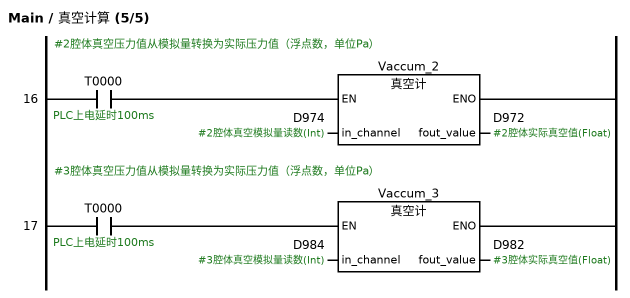
; [picture p24: Main / 真空计算, rungs 16-17]
; rung 16: #2腔体真空压力值从模拟量转换为实际压力值（浮点数，单位Pa）
LD T0000  ; PLC上电延时100ms
CALL Vaccum_2 : 真空计 (in_channel := D974, fout_value => D972)  ; #2腔体真空模拟量读数(Int), #2腔体实际真空值(Float)
; rung 17: #3腔体真空压力值从模拟量转换为实际压力值（浮点数，单位Pa）
LD T0000  ; PLC上电延时100ms
CALL Vaccum_3 : 真空计 (in_channel := D984, fout_value => D982)  ; #3腔体真空模拟量读数(Int), #3腔体实际真空值(Float)

### Section 整机复位

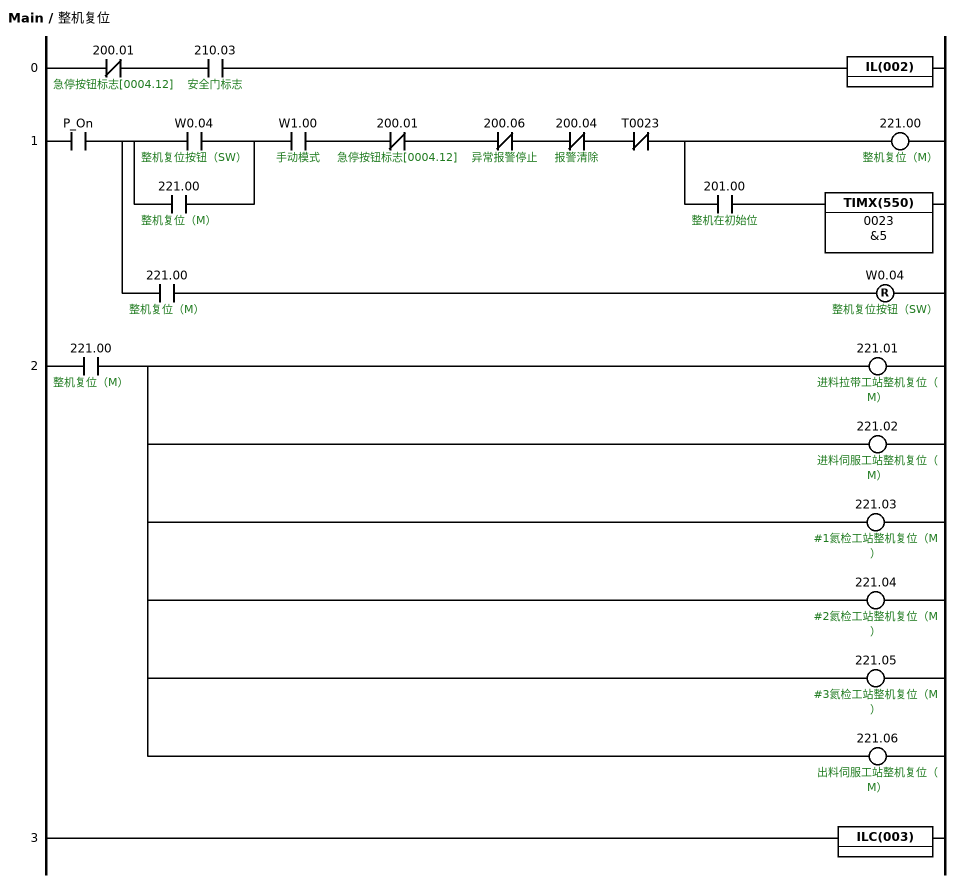
; rung 0
LDNOT 200.01  ; 急停按钮标志[0004.12]
AND 210.03  ; 安全门标志
IL(002)
; rung 1
LD P_On
OUT TR0
LD W0.04  ; 整机复位按钮（SW）
OR 221.00  ; 整机复位（M）
ANDLD
AND W1.00  ; 手动模式
ANDNOT 200.01  ; 急停按钮标志[0004.12]
ANDNOT 200.06  ; 异常报警停止
ANDNOT 200.04  ; 报警清除
ANDNOT T0023
OUT 221.00  ; 整机复位（M）
AND 201.00  ; 整机在初始位
TIMX(550) 0023 &5
LD TR0
AND 221.00  ; 整机复位（M）
RSET W0.04  ; 整机复位按钮（SW）
; rung 2
LD 221.00  ; 整机复位（M）
OUT 221.01  ; 进料拉带工站整机复位（M）
OUT 221.02  ; 进料伺服工站整机复位（M）
OUT 221.03  ; #1氦检工站整机复位（M）
OUT 221.04  ; #2氦检工站整机复位（M）
OUT 221.05  ; #3氦检工站整机复位（M）
OUT 221.06  ; 出料伺服工站整机复位（M）
; rung 3
ILC(003)

### Section 指示灯

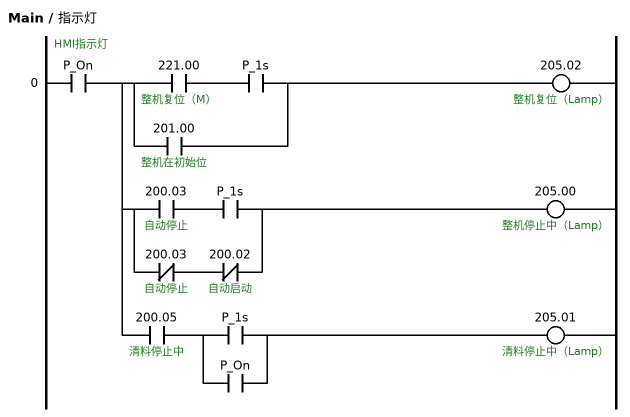
; rung 0: HMI指示灯
LD P_On
OUT TR0
LD 221.00  ; 整机复位（M）
AND P_1s
OR 201.00  ; 整机在初始位
ANDLD
OUT 205.02  ; 整机复位（Lamp）
LD TR0
LD 200.03  ; 自动停止
AND P_1s
LDNOT 200.03  ; 自动停止
ANDNOT 200.02  ; 自动启动
ORLD
ANDLD
OUT 205.00  ; 整机停止中（Lamp）
LD TR0
AND 200.05  ; 清料停止中
LD P_1s
OR P_On
ANDLD
OUT 205.01  ; 清料停止中（Lamp）

### Section 外部输出

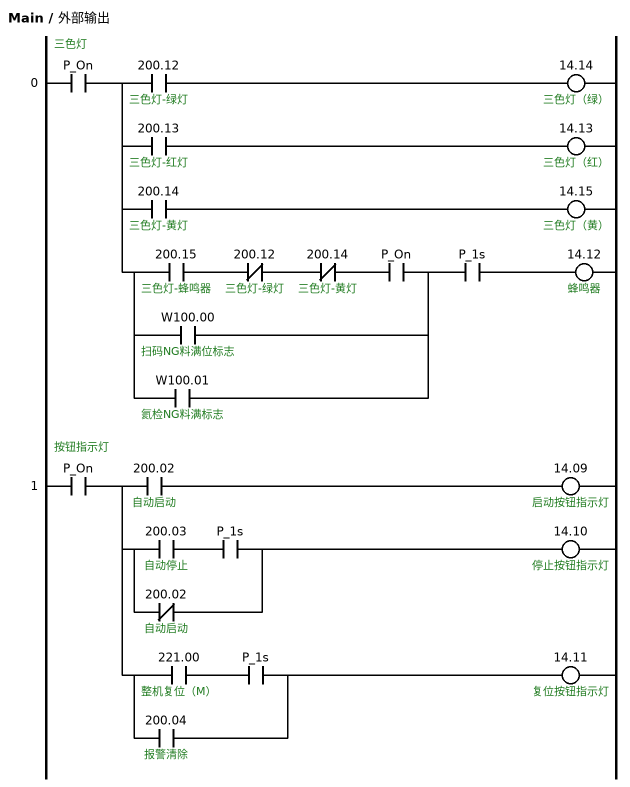
; rung 0: 三色灯
LD P_On
OUT TR0
AND 200.12  ; 三色灯-绿灯
OUT 14.14  ; 三色灯（绿）
LD TR0
AND 200.13  ; 三色灯-红灯
OUT 14.13  ; 三色灯（红）
LD TR0
AND 200.14  ; 三色灯-黄灯
OUT 14.15  ; 三色灯（黄）
LD TR0
LD 200.15  ; 三色灯-蜂鸣器
ANDNOT 200.12  ; 三色灯-绿灯
ANDNOT 200.14  ; 三色灯-黄灯
AND P_On
OR W100.00  ; 扫码NG料满位标志
OR W100.01  ; 氦检NG料满标志
ANDLD
AND P_1s
OUT 14.12  ; 蜂鸣器
; rung 1: 按钮指示灯
LD P_On
OUT TR0
AND 200.02  ; 自动启动
OUT 14.09  ; 启动按钮指示灯
LD TR0
LD 200.03  ; 自动停止
AND P_1s
ORNOT 200.02  ; 自动启动
ANDLD
OUT 14.10  ; 停止按钮指示灯
LD TR0
LD 221.00  ; 整机复位（M）
AND P_1s
OR 200.04  ; 报警清除
ANDLD
OUT 14.11  ; 复位按钮指示灯

### Section END
; rung 0
END(001)

## Program 进料拉带机构 (cyclic task 1)

### Section Main

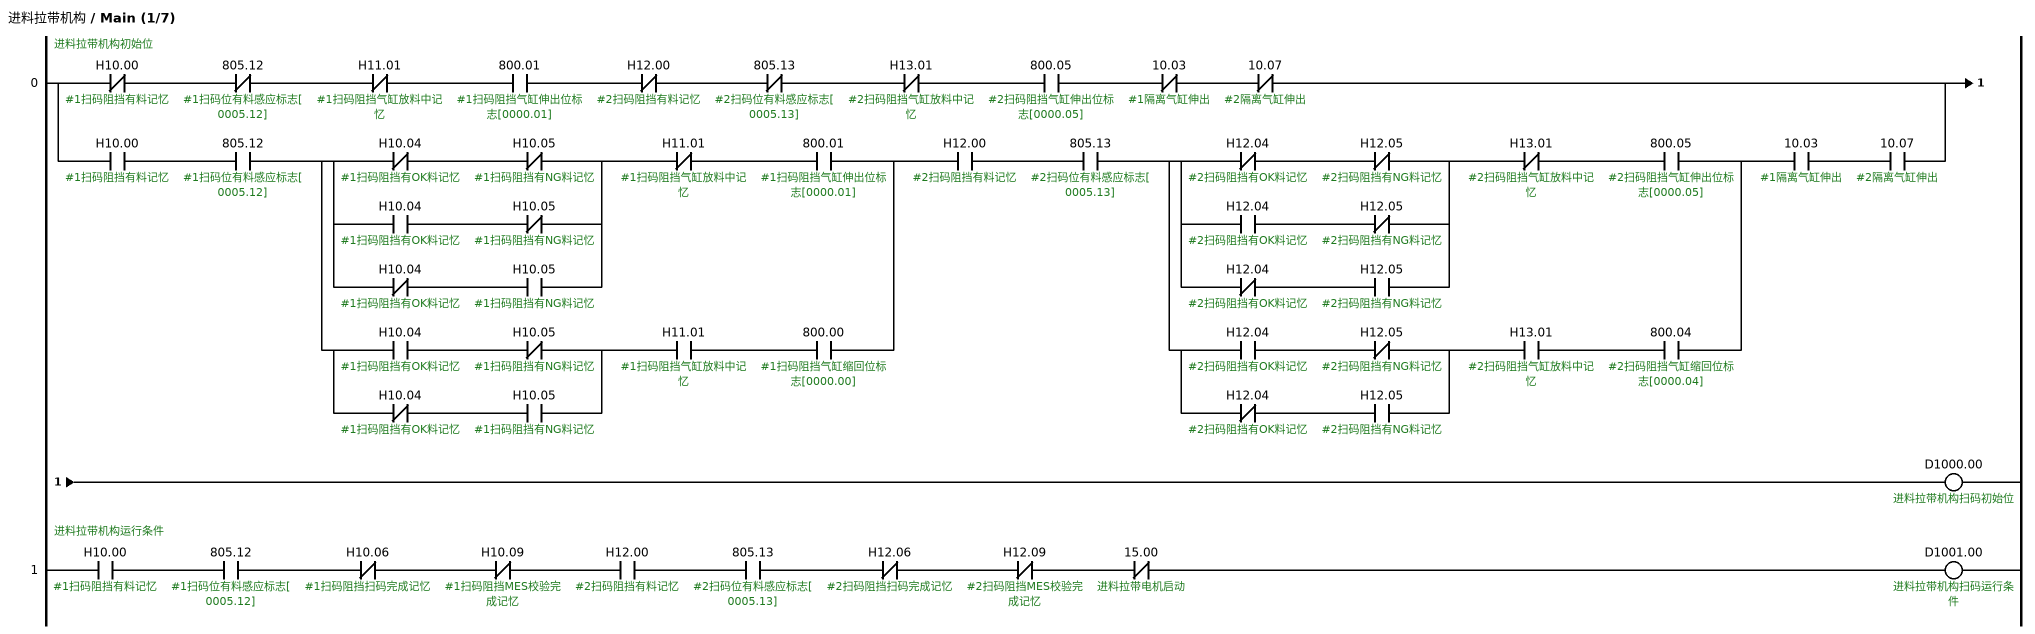
; rung 0: 进料拉带机构初始位
LDNOT H10.00  ; #1扫码阻挡有料记忆
ANDNOT 805.12  ; #1扫码位有料感应标志[0005.12]
ANDNOT H11.01  ; #1扫码阻挡气缸放料中记忆
AND 800.01  ; #1扫码阻挡气缸伸出位标志[0000.01]
ANDNOT H12.00  ; #2扫码阻挡有料记忆
ANDNOT 805.13  ; #2扫码位有料感应标志[0005.13]
ANDNOT H13.01  ; #2扫码阻挡气缸放料中记忆
AND 800.05  ; #2扫码阻挡气缸伸出位标志[0000.05]
ANDNOT 10.03  ; #1隔离气缸伸出
ANDNOT 10.07  ; #2隔离气缸伸出
LD H10.00  ; #1扫码阻挡有料记忆
AND 805.12  ; #1扫码位有料感应标志[0005.12]
LDNOT H10.04  ; #1扫码阻挡有OK料记忆
ANDNOT H10.05  ; #1扫码阻挡有NG料记忆
LD H10.04  ; #1扫码阻挡有OK料记忆
ANDNOT H10.05  ; #1扫码阻挡有NG料记忆
ORLD
LDNOT H10.04  ; #1扫码阻挡有OK料记忆
AND H10.05  ; #1扫码阻挡有NG料记忆
ORLD
ANDNOT H11.01  ; #1扫码阻挡气缸放料中记忆
AND 800.01  ; #1扫码阻挡气缸伸出位标志[0000.01]
LD H10.04  ; #1扫码阻挡有OK料记忆
ANDNOT H10.05  ; #1扫码阻挡有NG料记忆
LDNOT H10.04  ; #1扫码阻挡有OK料记忆
AND H10.05  ; #1扫码阻挡有NG料记忆
ORLD
AND H11.01  ; #1扫码阻挡气缸放料中记忆
AND 800.00  ; #1扫码阻挡气缸缩回位标志[0000.00]
ORLD
ANDLD
AND H12.00  ; #2扫码阻挡有料记忆
AND 805.13  ; #2扫码位有料感应标志[0005.13]
LDNOT H12.04  ; #2扫码阻挡有OK料记忆
ANDNOT H12.05  ; #2扫码阻挡有NG料记忆
LD H12.04  ; #2扫码阻挡有OK料记忆
ANDNOT H12.05  ; #2扫码阻挡有NG料记忆
ORLD
LDNOT H12.04  ; #2扫码阻挡有OK料记忆
AND H12.05  ; #2扫码阻挡有NG料记忆
ORLD
ANDNOT H13.01  ; #2扫码阻挡气缸放料中记忆
AND 800.05  ; #2扫码阻挡气缸伸出位标志[0000.05]
LD H12.04  ; #2扫码阻挡有OK料记忆
ANDNOT H12.05  ; #2扫码阻挡有NG料记忆
LDNOT H12.04  ; #2扫码阻挡有OK料记忆
AND H12.05  ; #2扫码阻挡有NG料记忆
ORLD
AND H13.01  ; #2扫码阻挡气缸放料中记忆
AND 800.04  ; #2扫码阻挡气缸缩回位标志[0000.04]
ORLD
ANDLD
AND 10.03  ; #1隔离气缸伸出
AND 10.07  ; #2隔离气缸伸出
ORLD
OUT D1000.00  ; 进料拉带机构扫码初始位
; rung 1: 进料拉带机构运行条件
LD H10.00  ; #1扫码阻挡有料记忆
AND 805.12  ; #1扫码位有料感应标志[0005.12]
ANDNOT H10.06  ; #1扫码阻挡扫码完成记忆
ANDNOT H10.09  ; #1扫码阻挡MES校验完成记忆
AND H12.00  ; #2扫码阻挡有料记忆
AND 805.13  ; #2扫码位有料感应标志[0005.13]
ANDNOT H12.06  ; #2扫码阻挡扫码完成记忆
ANDNOT H12.09  ; #2扫码阻挡MES校验完成记忆
ANDNOT 15.00  ; 进料拉带电机启动
OUT D1001.00  ; 进料拉带机构扫码运行条件

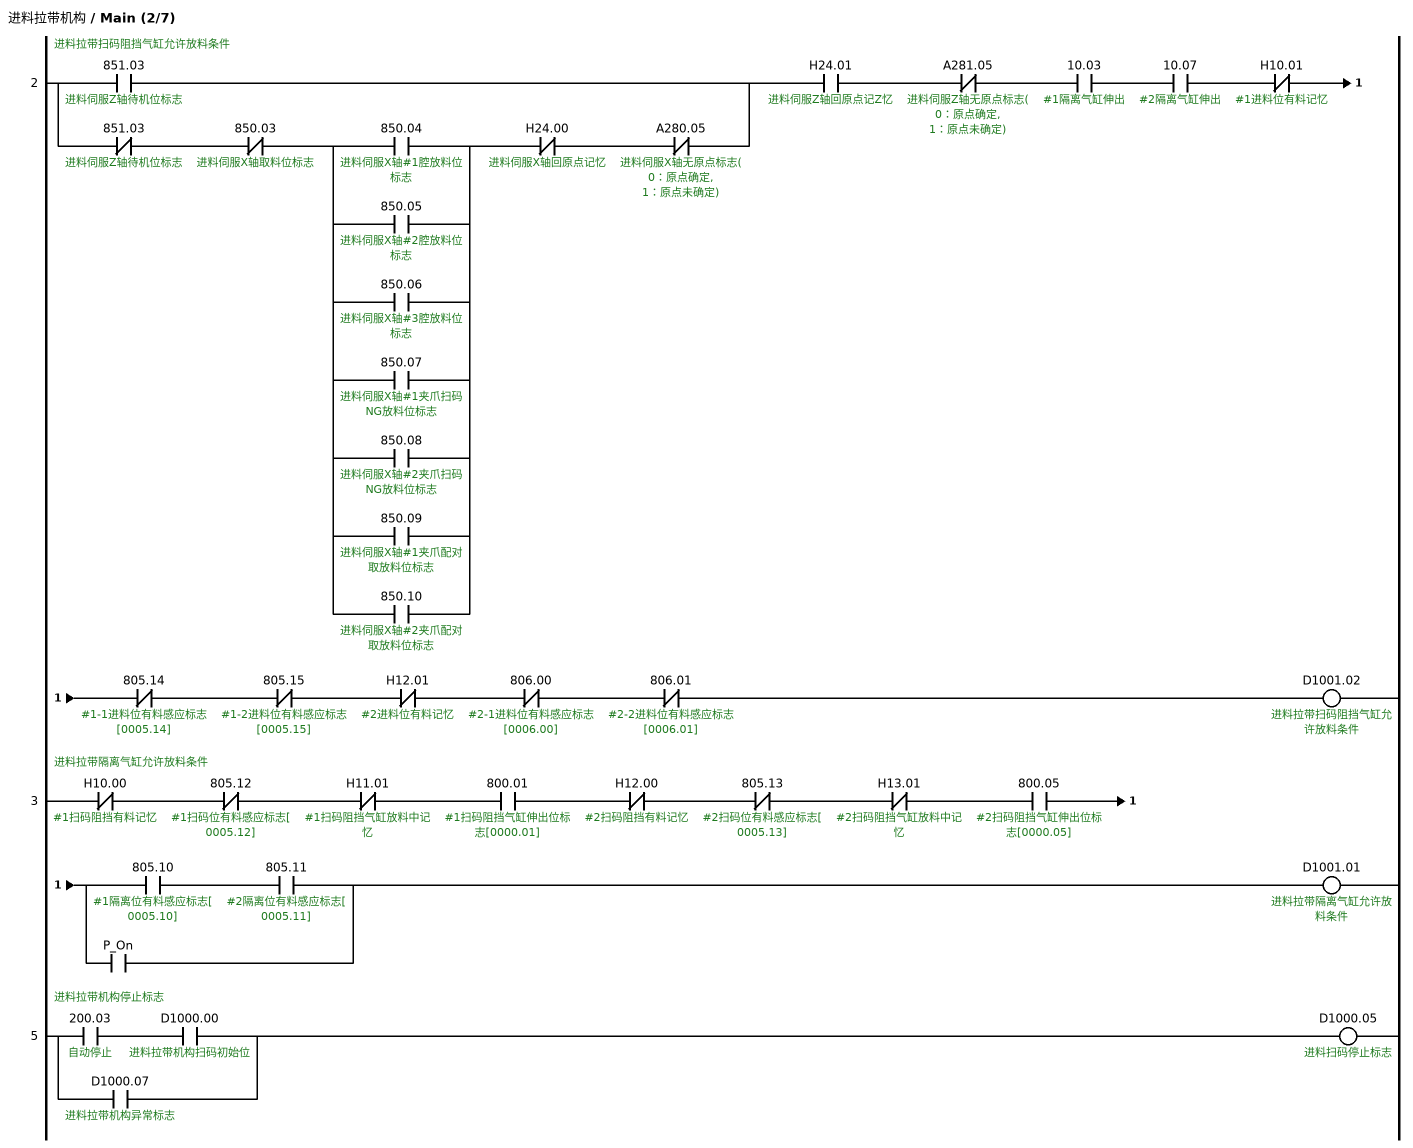
; rung 2: 进料拉带扫码阻挡气缸允许放料条件
LD 851.03  ; 进料伺服Z轴待机位标志
LDNOT 851.03  ; 进料伺服Z轴待机位标志
ANDNOT 850.03  ; 进料伺服X轴取料位标志
LD 850.04  ; 进料伺服X轴#1腔放料位标志
OR 850.05  ; 进料伺服X轴#2腔放料位标志
OR 850.06  ; 进料伺服X轴#3腔放料位标志
OR 850.07  ; 进料伺服X轴#1夹爪扫码NG放料位标志
OR 850.08  ; 进料伺服X轴#2夹爪扫码NG放料位标志
OR 850.09  ; 进料伺服X轴#1夹爪配对取放料位标志
OR 850.10  ; 进料伺服X轴#2夹爪配对取放料位标志
ANDLD
ANDNOT H24.00  ; 进料伺服X轴回原点记忆
ANDNOT A280.05  ; 进料伺服X轴无原点标志(0：原点确定,1：原点未确定)
ORLD
AND H24.01  ; 进料伺服Z轴回原点记Z忆
ANDNOT A281.05  ; 进料伺服Z轴无原点标志(0：原点确定,1：原点未确定)
AND 10.03  ; #1隔离气缸伸出
AND 10.07  ; #2隔离气缸伸出
ANDNOT H10.01  ; #1进料位有料记忆
ANDNOT 805.14  ; #1-1进料位有料感应标志[0005.14]
ANDNOT 805.15  ; #1-2进料位有料感应标志[0005.15]
ANDNOT H12.01  ; #2进料位有料记忆
ANDNOT 806.00  ; #2-1进料位有料感应标志[0006.00]
ANDNOT 806.01  ; #2-2进料位有料感应标志[0006.01]
OUT D1001.02  ; 进料拉带扫码阻挡气缸允许放料条件
; rung 3: 进料拉带隔离气缸允许放料条件
LDNOT H10.00  ; #1扫码阻挡有料记忆
ANDNOT 805.12  ; #1扫码位有料感应标志[0005.12]
ANDNOT H11.01  ; #1扫码阻挡气缸放料中记忆
AND 800.01  ; #1扫码阻挡气缸伸出位标志[0000.01]
ANDNOT H12.00  ; #2扫码阻挡有料记忆
ANDNOT 805.13  ; #2扫码位有料感应标志[0005.13]
ANDNOT H13.01  ; #2扫码阻挡气缸放料中记忆
AND 800.05  ; #2扫码阻挡气缸伸出位标志[0000.05]
LD 805.10  ; #1隔离位有料感应标志[0005.10]
AND 805.11  ; #2隔离位有料感应标志[0005.11]
OR P_On
ANDLD
OUT D1001.01  ; 进料拉带隔离气缸允许放料条件
; rung 4: 进料拉带上料位允许抓料条件
; rung 5: 进料拉带机构停止标志
LD 200.03  ; 自动停止
AND D1000.00  ; 进料拉带机构扫码初始位
OR D1000.07  ; 进料拉带机构异常标志
OUT D1000.05  ; 进料扫码停止标志

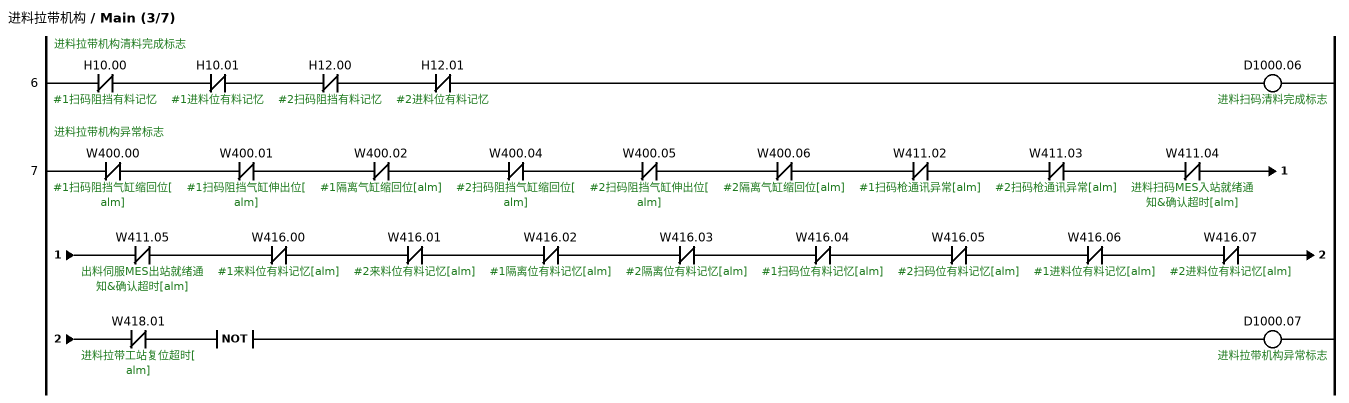
; rung 6: 进料拉带机构清料完成标志
LDNOT H10.00  ; #1扫码阻挡有料记忆
ANDNOT H10.01  ; #1进料位有料记忆
ANDNOT H12.00  ; #2扫码阻挡有料记忆
ANDNOT H12.01  ; #2进料位有料记忆
OUT D1000.06  ; 进料扫码清料完成标志
; rung 7: 进料拉带机构异常标志
LDNOT W400.00  ; #1扫码阻挡气缸缩回位[alm]
ANDNOT W400.01  ; #1扫码阻挡气缸伸出位[alm]
ANDNOT W400.02  ; #1隔离气缸缩回位[alm]
ANDNOT W400.04  ; #2扫码阻挡气缸缩回位[alm]
ANDNOT W400.05  ; #2扫码阻挡气缸伸出位[alm]
ANDNOT W400.06  ; #2隔离气缸缩回位[alm]
ANDNOT W411.02  ; #1扫码枪通讯异常[alm]
ANDNOT W411.03  ; #2扫码枪通讯异常[alm]
ANDNOT W411.04  ; 进料扫码MES入站就绪通知&确认超时[alm]
ANDNOT W411.05  ; 出料伺服MES出站就绪通知&确认超时[alm]
ANDNOT W416.00  ; #1来料位有料记忆[alm]
ANDNOT W416.01  ; #2来料位有料记忆[alm]
ANDNOT W416.02  ; #1隔离位有料记忆[alm]
ANDNOT W416.03  ; #2隔离位有料记忆[alm]
ANDNOT W416.04  ; #1扫码位有料记忆[alm]
ANDNOT W416.05  ; #2扫码位有料记忆[alm]
ANDNOT W416.06  ; #1进料位有料记忆[alm]
ANDNOT W416.07  ; #2进料位有料记忆[alm]
ANDNOT W418.01  ; 进料拉带工站复位超时[alm]
NOT(520)
OUT D1000.07  ; 进料拉带机构异常标志

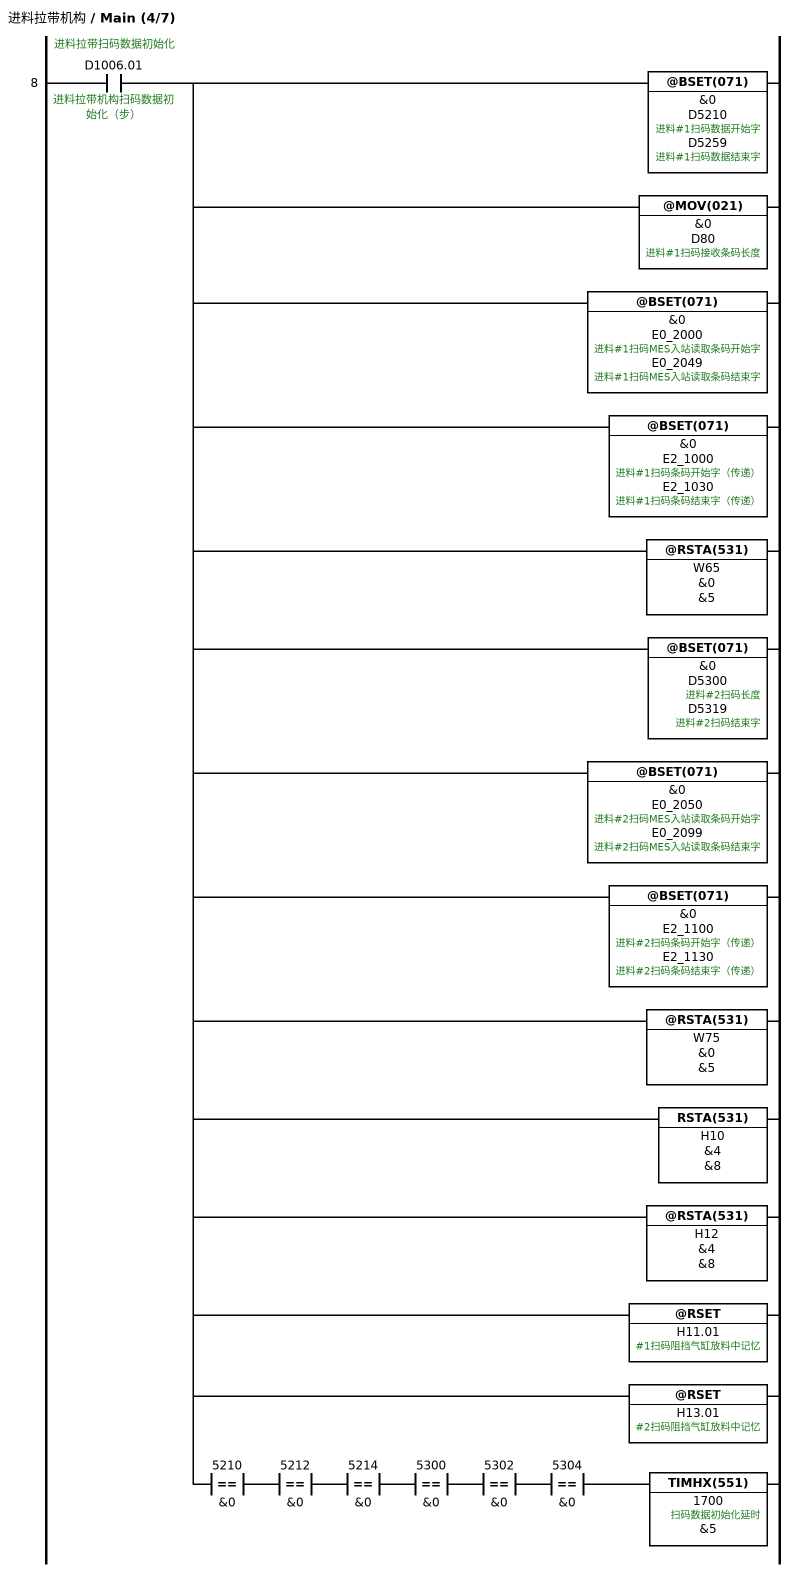
; rung 8: 进料拉带扫码数据初始化
LD D1006.01  ; 进料拉带机构扫码数据初始化（步）
@BSET(071) &0 D5210 D5259  ; 进料#1扫码数据开始字, 进料#1扫码数据结束字
@MOV(021) &0 D80  ; 进料#1扫码接收条码长度
@BSET(071) &0 E0_2000 E0_2049  ; 进料#1扫码MES入站读取条码开始字, 进料#1扫码MES入站读取条码结束字
@BSET(071) &0 E2_1000 E2_1030  ; 进料#1扫码条码开始字（传递）, 进料#1扫码条码结束字（传递）
@RSTA(531) W65 &0 &5
@BSET(071) &0 D5300 D5319  ; 进料#2扫码长度, 进料#2扫码结束字
@BSET(071) &0 E0_2050 E0_2099  ; 进料#2扫码MES入站读取条码开始字, 进料#2扫码MES入站读取条码结束字
@BSET(071) &0 E2_1100 E2_1130  ; 进料#2扫码条码开始字（传递）, 进料#2扫码条码结束字（传递）
@RSTA(531) W75 &0 &5
RSTA(531) H10 &4 &8
@RSTA(531) H12 &4 &8
@RSET H11.01  ; #1扫码阻挡气缸放料中记忆
@RSET H13.01  ; #2扫码阻挡气缸放料中记忆
AND=L(301) 5210 &0
AND=L(301) 5212 &0
AND=L(301) 5214 &0
AND=L(301) 5300 &0
AND=L(301) 5302 &0
AND=L(301) 5304 &0
TIMHX(551) 1700 &5  ; 扫码数据初始化延时

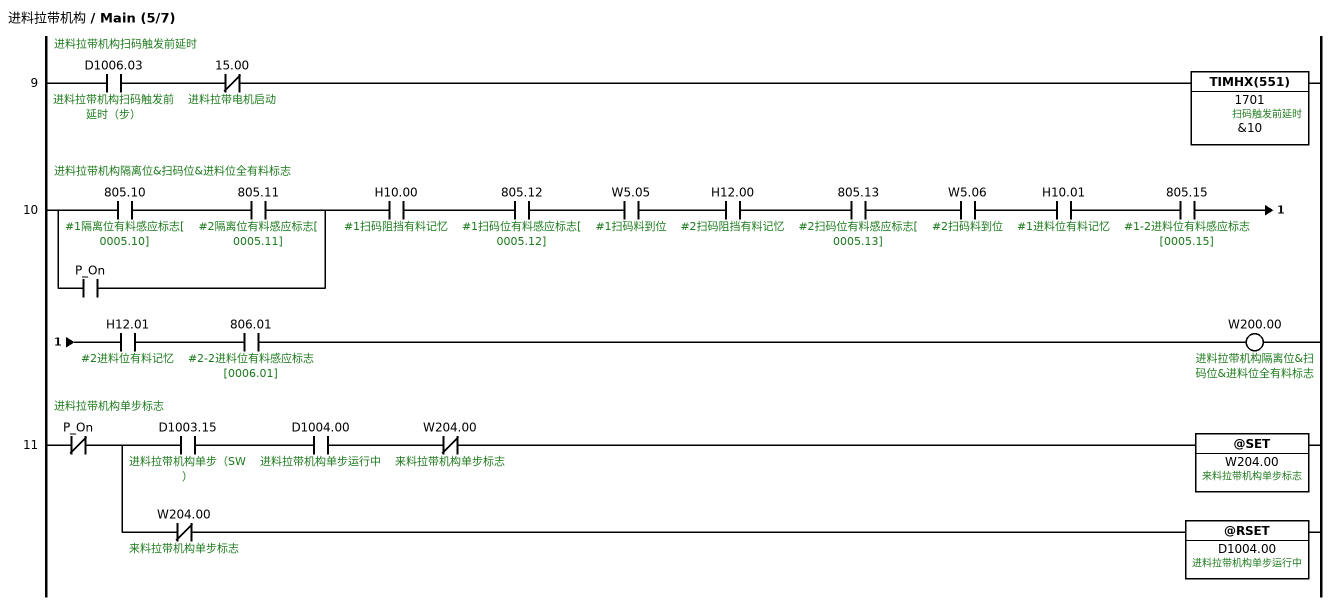
; rung 9: 进料拉带机构扫码触发前延时
LD D1006.03  ; 进料拉带机构扫码触发前延时（步）
ANDNOT 15.00  ; 进料拉带电机启动
TIMHX(551) 1701 &10  ; 扫码触发前延时
; rung 10: 进料拉带机构隔离位&扫码位&进料位全有料标志
LD 805.10  ; #1隔离位有料感应标志[0005.10]
AND 805.11  ; #2隔离位有料感应标志[0005.11]
OR P_On
AND H10.00  ; #1扫码阻挡有料记忆
AND 805.12  ; #1扫码位有料感应标志[0005.12]
AND W5.05  ; #1扫码料到位
AND H12.00  ; #2扫码阻挡有料记忆
AND 805.13  ; #2扫码位有料感应标志[0005.13]
AND W5.06  ; #2扫码料到位
AND H10.01  ; #1进料位有料记忆
AND 805.15  ; #1-2进料位有料感应标志[0005.15]
AND H12.01  ; #2进料位有料记忆
AND 806.01  ; #2-2进料位有料感应标志[0006.01]
OUT W200.00  ; 进料拉带机构隔离位&扫码位&进料位全有料标志
; rung 11: 进料拉带机构单步标志
LDNOT P_On
OUT TR0
AND D1003.15  ; 进料拉带机构单步（SW）
AND D1004.00  ; 进料拉带机构单步运行中
ANDNOT W204.00  ; 来料拉带机构单步标志
@SET W204.00  ; 来料拉带机构单步标志
LD TR0
ANDNOT W204.00  ; 来料拉带机构单步标志
@RSET D1004.00  ; 进料拉带机构单步运行中

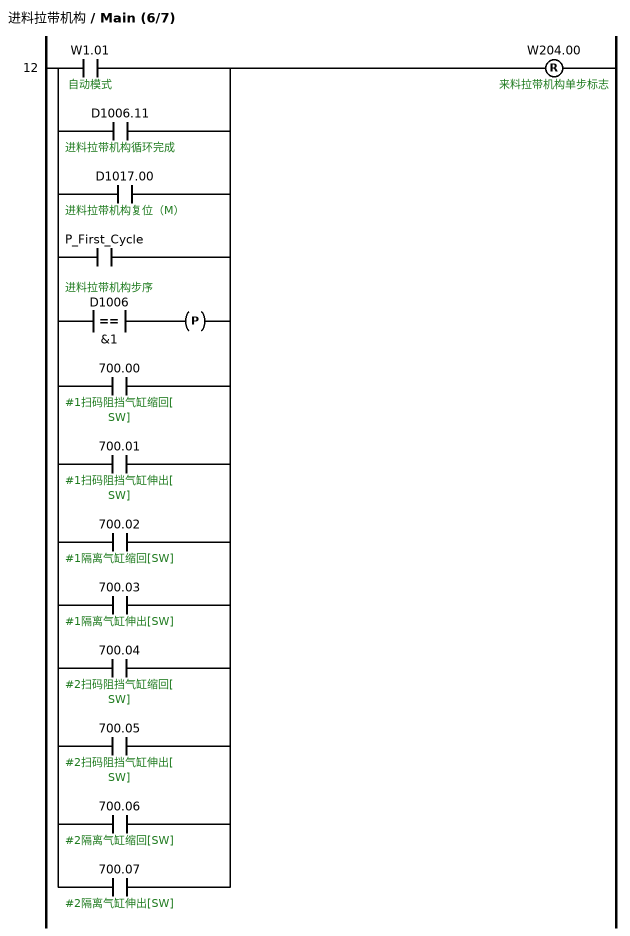
; rung 12
LD W1.01  ; 自动模式
OR D1006.11  ; 进料拉带机构循环完成
OR D1017.00  ; 进料拉带机构复位（M）
OR P_First_Cycle
LD=(300) D1006 &1  ; 进料拉带机构步序
UP(521)
ORLD
OR 700.00  ; #1扫码阻挡气缸缩回[SW]
OR 700.01  ; #1扫码阻挡气缸伸出[SW]
OR 700.02  ; #1隔离气缸缩回[SW]
OR 700.03  ; #1隔离气缸伸出[SW]
OR 700.04  ; #2扫码阻挡气缸缩回[SW]
OR 700.05  ; #2扫码阻挡气缸伸出[SW]
OR 700.06  ; #2隔离气缸缩回[SW]
OR 700.07  ; #2隔离气缸伸出[SW]
RSET W204.00  ; 来料拉带机构单步标志

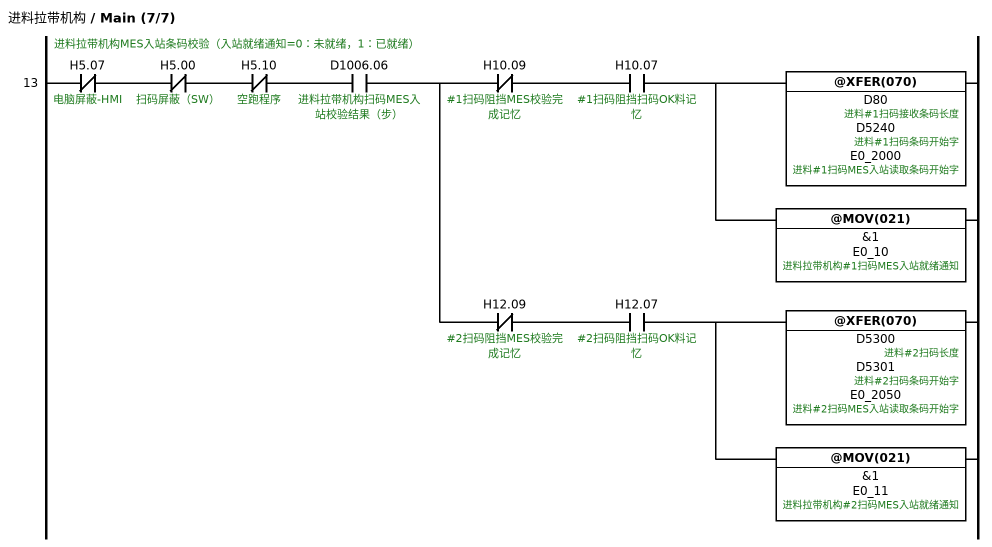
; rung 13: 进料拉带机构MES入站条码校验（入站就绪通知=0：未就绪，1：已就绪）
LDNOT H5.07  ; 电脑屏蔽-HMI
ANDNOT H5.00  ; 扫码屏蔽（SW）
ANDNOT H5.10  ; 空跑程序
AND D1006.06  ; 进料拉带机构扫码MES入站校验结果（步）
OUT TR0
ANDNOT H10.09  ; #1扫码阻挡MES校验完成记忆
AND H10.07  ; #1扫码阻挡扫码OK料记忆
@XFER(070) D80 D5240 E0_2000  ; 进料#1扫码接收条码长度, 进料#1扫码条码开始字, 进料#1扫码MES入站读取条码开始字
@MOV(021) &1 E0_10  ; 进料拉带机构#1扫码MES入站就绪通知
LD TR0
ANDNOT H12.09  ; #2扫码阻挡MES校验完成记忆
AND H12.07  ; #2扫码阻挡扫码OK料记忆
@XFER(070) D5300 D5301 E0_2050  ; 进料#2扫码长度, 进料#2扫码条码开始字, 进料#2扫码MES入站读取条码开始字
@MOV(021) &1 E0_11  ; 进料拉带机构#2扫码MES入站就绪通知

### Section 进料手动

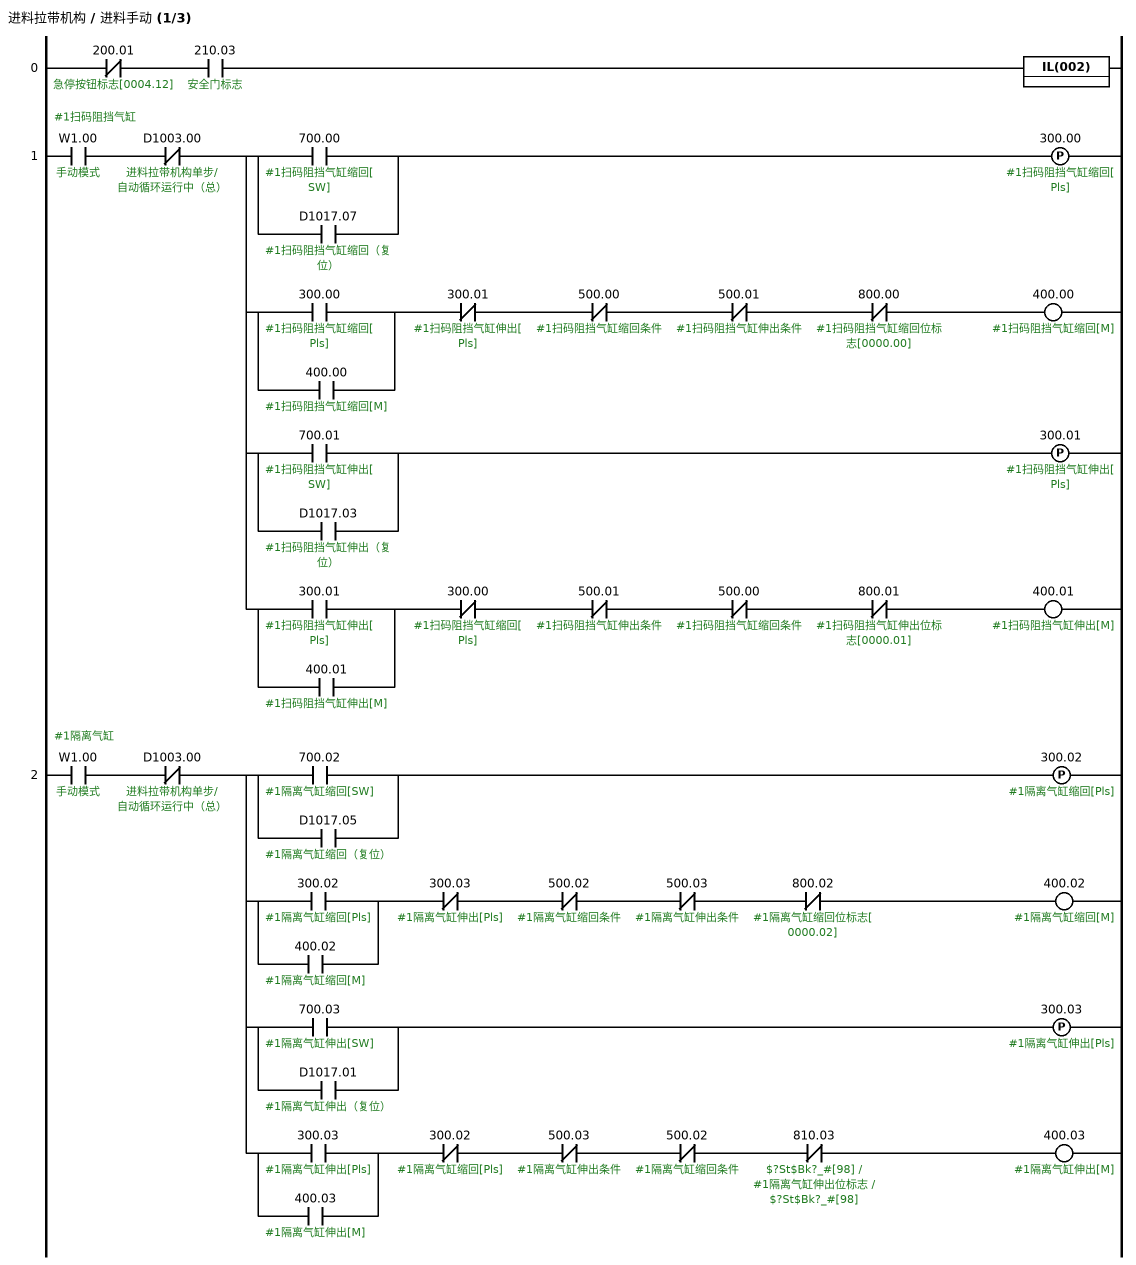
; rung 0
LDNOT 200.01  ; 急停按钮标志[0004.12]
AND 210.03  ; 安全门标志
IL(002)
; rung 1: #1扫码阻挡气缸
LD W1.00  ; 手动模式
ANDNOT D1003.00  ; 进料拉带机构单步/自动循环运行中（总）
OUT TR0
LD 700.00  ; #1扫码阻挡气缸缩回[SW]
OR D1017.07  ; #1扫码阻挡气缸缩回（复位）
ANDLD
DIFU(013) 300.00  ; #1扫码阻挡气缸缩回[Pls]
LD TR0
LD 300.00  ; #1扫码阻挡气缸缩回[Pls]
OR 400.00  ; #1扫码阻挡气缸缩回[M]
ANDLD
ANDNOT 300.01  ; #1扫码阻挡气缸伸出[Pls]
ANDNOT 500.00  ; #1扫码阻挡气缸缩回条件
ANDNOT 500.01  ; #1扫码阻挡气缸伸出条件
ANDNOT 800.00  ; #1扫码阻挡气缸缩回位标志[0000.00]
OUT 400.00  ; #1扫码阻挡气缸缩回[M]
LD TR0
LD 700.01  ; #1扫码阻挡气缸伸出[SW]
OR D1017.03  ; #1扫码阻挡气缸伸出（复位）
ANDLD
DIFU(013) 300.01  ; #1扫码阻挡气缸伸出[Pls]
LD TR0
LD 300.01  ; #1扫码阻挡气缸伸出[Pls]
OR 400.01  ; #1扫码阻挡气缸伸出[M]
ANDLD
ANDNOT 300.00  ; #1扫码阻挡气缸缩回[Pls]
ANDNOT 500.01  ; #1扫码阻挡气缸伸出条件
ANDNOT 500.00  ; #1扫码阻挡气缸缩回条件
ANDNOT 800.01  ; #1扫码阻挡气缸伸出位标志[0000.01]
OUT 400.01  ; #1扫码阻挡气缸伸出[M]
; rung 2: #1隔离气缸
LD W1.00  ; 手动模式
ANDNOT D1003.00  ; 进料拉带机构单步/自动循环运行中（总）
OUT TR0
LD 700.02  ; #1隔离气缸缩回[SW]
OR D1017.05  ; #1隔离气缸缩回（复位）
ANDLD
DIFU(013) 300.02  ; #1隔离气缸缩回[Pls]
LD TR0
LD 300.02  ; #1隔离气缸缩回[Pls]
OR 400.02  ; #1隔离气缸缩回[M]
ANDLD
ANDNOT 300.03  ; #1隔离气缸伸出[Pls]
ANDNOT 500.02  ; #1隔离气缸缩回条件
ANDNOT 500.03  ; #1隔离气缸伸出条件
ANDNOT 800.02  ; #1隔离气缸缩回位标志[0000.02]
OUT 400.02  ; #1隔离气缸缩回[M]
LD TR0
LD 700.03  ; #1隔离气缸伸出[SW]
OR D1017.01  ; #1隔离气缸伸出（复位）
ANDLD
DIFU(013) 300.03  ; #1隔离气缸伸出[Pls]
LD TR0
LD 300.03  ; #1隔离气缸伸出[Pls]
OR 400.03  ; #1隔离气缸伸出[M]
ANDLD
ANDNOT 300.02  ; #1隔离气缸缩回[Pls]
ANDNOT 500.03  ; #1隔离气缸伸出条件
ANDNOT 500.02  ; #1隔离气缸缩回条件
ANDNOT 810.03  ; $?St$Bk?_#[98] / #1隔离气缸伸出位标志 / $?St$Bk?_#[98]
OUT 400.03  ; #1隔离气缸伸出[M]

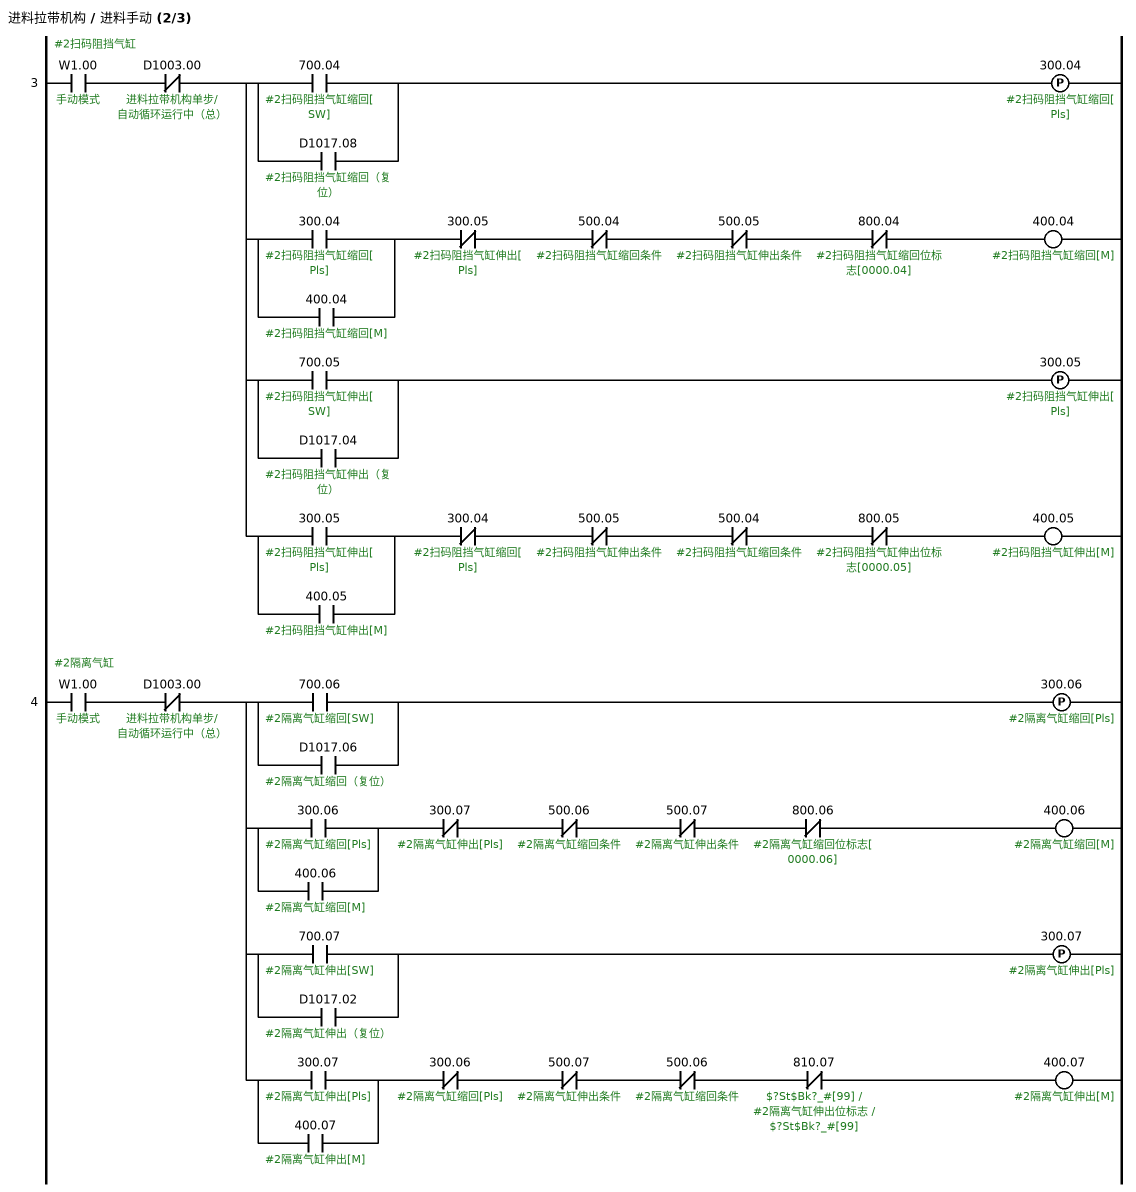
; rung 3: #2扫码阻挡气缸
LD W1.00  ; 手动模式
ANDNOT D1003.00  ; 进料拉带机构单步/自动循环运行中（总）
OUT TR0
LD 700.04  ; #2扫码阻挡气缸缩回[SW]
OR D1017.08  ; #2扫码阻挡气缸缩回（复位）
ANDLD
DIFU(013) 300.04  ; #2扫码阻挡气缸缩回[Pls]
LD TR0
LD 300.04  ; #2扫码阻挡气缸缩回[Pls]
OR 400.04  ; #2扫码阻挡气缸缩回[M]
ANDLD
ANDNOT 300.05  ; #2扫码阻挡气缸伸出[Pls]
ANDNOT 500.04  ; #2扫码阻挡气缸缩回条件
ANDNOT 500.05  ; #2扫码阻挡气缸伸出条件
ANDNOT 800.04  ; #2扫码阻挡气缸缩回位标志[0000.04]
OUT 400.04  ; #2扫码阻挡气缸缩回[M]
LD TR0
LD 700.05  ; #2扫码阻挡气缸伸出[SW]
OR D1017.04  ; #2扫码阻挡气缸伸出（复位）
ANDLD
DIFU(013) 300.05  ; #2扫码阻挡气缸伸出[Pls]
LD TR0
LD 300.05  ; #2扫码阻挡气缸伸出[Pls]
OR 400.05  ; #2扫码阻挡气缸伸出[M]
ANDLD
ANDNOT 300.04  ; #2扫码阻挡气缸缩回[Pls]
ANDNOT 500.05  ; #2扫码阻挡气缸伸出条件
ANDNOT 500.04  ; #2扫码阻挡气缸缩回条件
ANDNOT 800.05  ; #2扫码阻挡气缸伸出位标志[0000.05]
OUT 400.05  ; #2扫码阻挡气缸伸出[M]
; rung 4: #2隔离气缸
LD W1.00  ; 手动模式
ANDNOT D1003.00  ; 进料拉带机构单步/自动循环运行中（总）
OUT TR0
LD 700.06  ; #2隔离气缸缩回[SW]
OR D1017.06  ; #2隔离气缸缩回（复位）
ANDLD
DIFU(013) 300.06  ; #2隔离气缸缩回[Pls]
LD TR0
LD 300.06  ; #2隔离气缸缩回[Pls]
OR 400.06  ; #2隔离气缸缩回[M]
ANDLD
ANDNOT 300.07  ; #2隔离气缸伸出[Pls]
ANDNOT 500.06  ; #2隔离气缸缩回条件
ANDNOT 500.07  ; #2隔离气缸伸出条件
ANDNOT 800.06  ; #2隔离气缸缩回位标志[0000.06]
OUT 400.06  ; #2隔离气缸缩回[M]
LD TR0
LD 700.07  ; #2隔离气缸伸出[SW]
OR D1017.02  ; #2隔离气缸伸出（复位）
ANDLD
DIFU(013) 300.07  ; #2隔离气缸伸出[Pls]
LD TR0
LD 300.07  ; #2隔离气缸伸出[Pls]
OR 400.07  ; #2隔离气缸伸出[M]
ANDLD
ANDNOT 300.06  ; #2隔离气缸缩回[Pls]
ANDNOT 500.07  ; #2隔离气缸伸出条件
ANDNOT 500.06  ; #2隔离气缸缩回条件
ANDNOT 810.07  ; $?St$Bk?_#[99] / #2隔离气缸伸出位标志 / $?St$Bk?_#[99]
OUT 400.07  ; #2隔离气缸伸出[M]

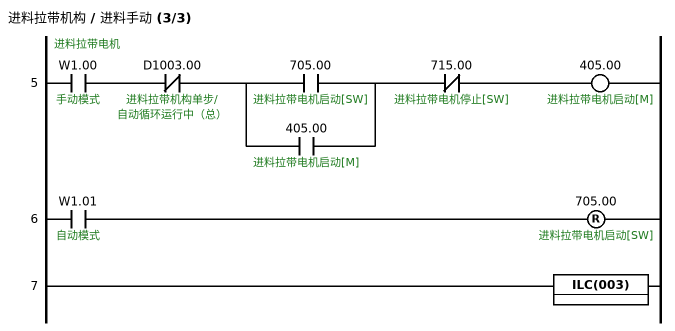
; rung 5: 进料拉带电机
LD W1.00  ; 手动模式
ANDNOT D1003.00  ; 进料拉带机构单步/自动循环运行中（总）
LD 705.00  ; 进料拉带电机启动[SW]
OR 405.00  ; 进料拉带电机启动[M]
ANDLD
ANDNOT 715.00  ; 进料拉带电机停止[SW]
OUT 405.00  ; 进料拉带电机启动[M]
; rung 6
LD W1.01  ; 自动模式
RSET 705.00  ; 进料拉带电机启动[SW]
; rung 7
ILC(003)

### Section 进料自动

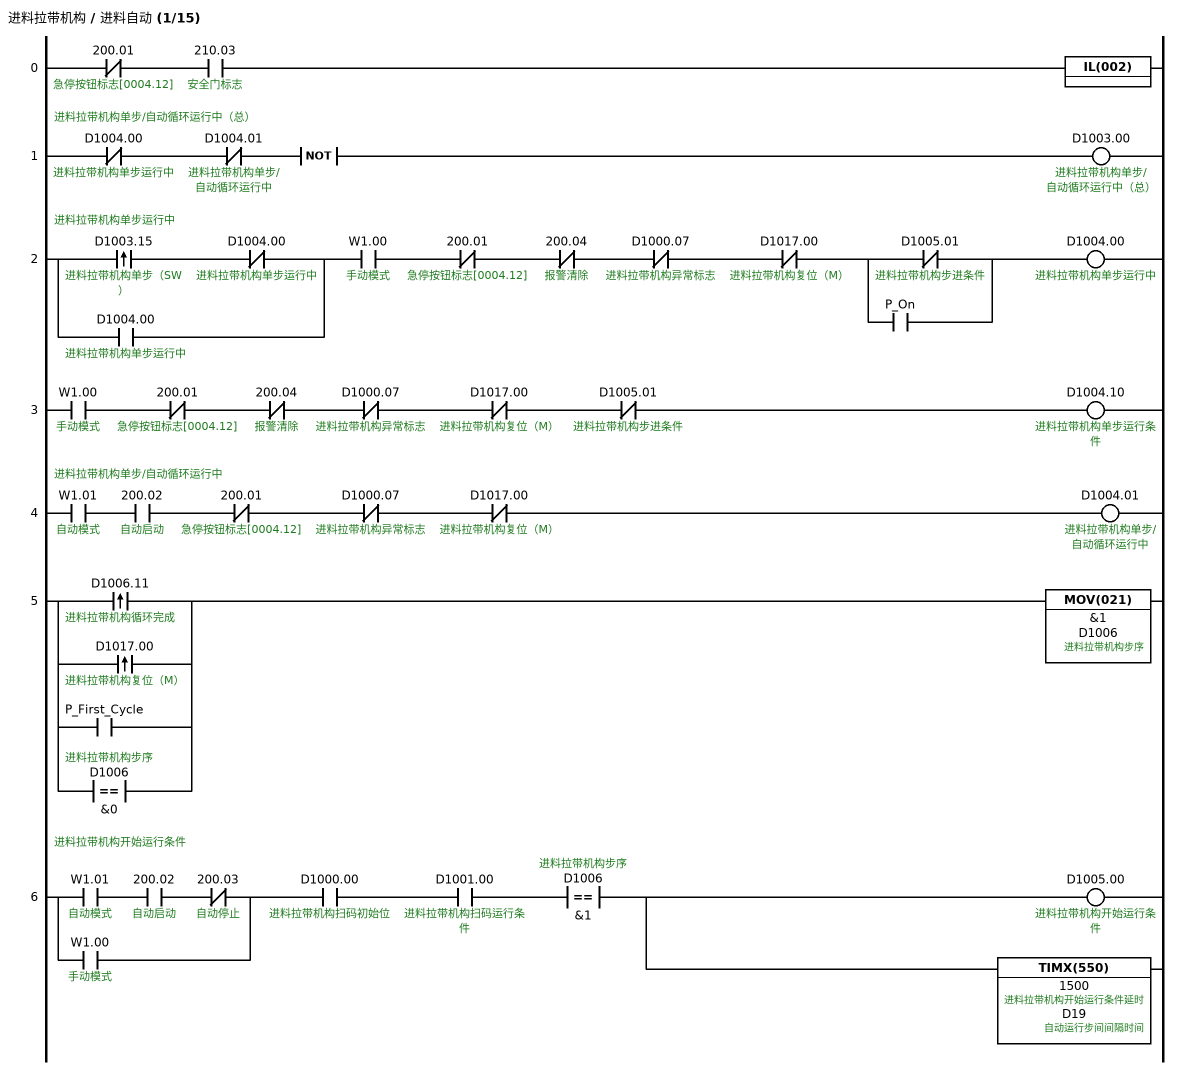
; rung 0
LDNOT 200.01  ; 急停按钮标志[0004.12]
AND 210.03  ; 安全门标志
IL(002)
; rung 1: 进料拉带机构单步/自动循环运行中（总）
LDNOT D1004.00  ; 进料拉带机构单步运行中
ANDNOT D1004.01  ; 进料拉带机构单步/自动循环运行中
NOT(520)
OUT D1003.00  ; 进料拉带机构单步/自动循环运行中（总）
; rung 2: 进料拉带机构单步运行中
@LD D1003.15  ; 进料拉带机构单步（SW）
ANDNOT D1004.00  ; 进料拉带机构单步运行中
OR D1004.00  ; 进料拉带机构单步运行中
AND W1.00  ; 手动模式
ANDNOT 200.01  ; 急停按钮标志[0004.12]
ANDNOT 200.04  ; 报警清除
ANDNOT D1000.07  ; 进料拉带机构异常标志
ANDNOT D1017.00  ; 进料拉带机构复位（M）
LDNOT D1005.01  ; 进料拉带机构步进条件
OR P_On
ANDLD
OUT D1004.00  ; 进料拉带机构单步运行中
; rung 3
LD W1.00  ; 手动模式
ANDNOT 200.01  ; 急停按钮标志[0004.12]
ANDNOT 200.04  ; 报警清除
ANDNOT D1000.07  ; 进料拉带机构异常标志
ANDNOT D1017.00  ; 进料拉带机构复位（M）
ANDNOT D1005.01  ; 进料拉带机构步进条件
OUT D1004.10  ; 进料拉带机构单步运行条件
; rung 4: 进料拉带机构单步/自动循环运行中
LD W1.01  ; 自动模式
AND 200.02  ; 自动启动
ANDNOT 200.01  ; 急停按钮标志[0004.12]
ANDNOT D1000.07  ; 进料拉带机构异常标志
ANDNOT D1017.00  ; 进料拉带机构复位（M）
OUT D1004.01  ; 进料拉带机构单步/自动循环运行中
; rung 5
@LD D1006.11  ; 进料拉带机构循环完成
@OR D1017.00  ; 进料拉带机构复位（M）
OR P_First_Cycle
OR=(300) D1006 &0  ; 进料拉带机构步序
MOV(021) &1 D1006  ; 进料拉带机构步序
; rung 6: 进料拉带机构开始运行条件
LD W1.01  ; 自动模式
AND 200.02  ; 自动启动
ANDNOT 200.03  ; 自动停止
OR W1.00  ; 手动模式
AND D1000.00  ; 进料拉带机构扫码初始位
AND D1001.00  ; 进料拉带机构扫码运行条件
AND=(300) D1006 &1  ; 进料拉带机构步序
OUT D1005.00  ; 进料拉带机构开始运行条件
TIMX(550) 1500 D19  ; 自动运行步间间隔时间, 进料拉带机构开始运行条件延时

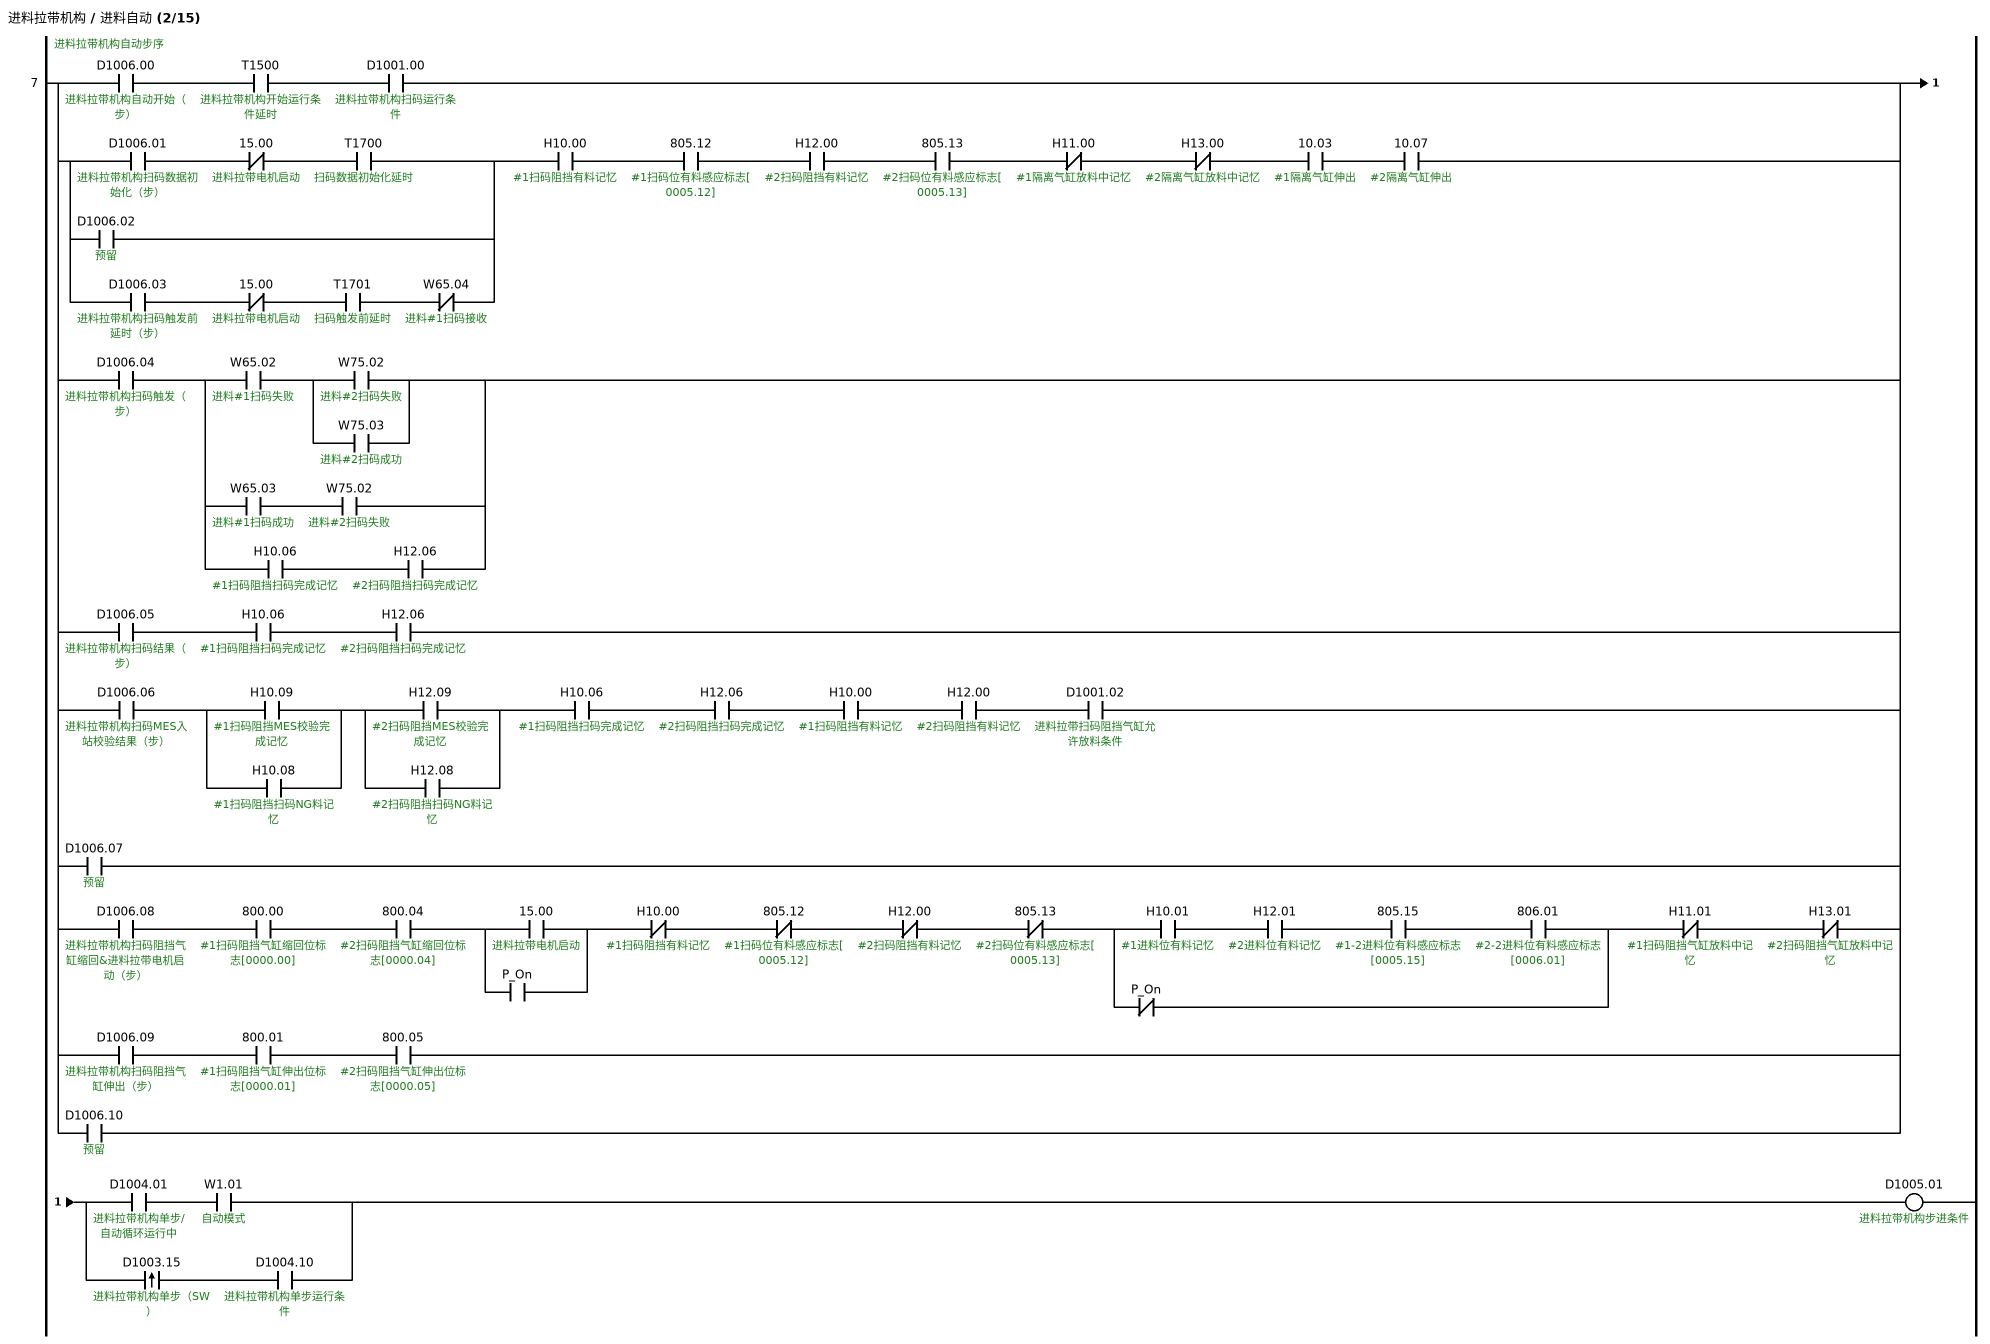
; rung 7: 进料拉带机构自动步序
LD D1006.00  ; 进料拉带机构自动开始（步）
AND T1500  ; 进料拉带机构开始运行条件延时
AND D1001.00  ; 进料拉带机构扫码运行条件
LD D1006.01  ; 进料拉带机构扫码数据初始化（步）
ANDNOT 15.00  ; 进料拉带电机启动
AND T1700  ; 扫码数据初始化延时
OR D1006.02  ; 预留
LD D1006.03  ; 进料拉带机构扫码触发前延时（步）
ANDNOT 15.00  ; 进料拉带电机启动
AND T1701  ; 扫码触发前延时
ANDNOT W65.04  ; 进料#1扫码接收
ORLD
AND H10.00  ; #1扫码阻挡有料记忆
AND 805.12  ; #1扫码位有料感应标志[0005.12]
AND H12.00  ; #2扫码阻挡有料记忆
AND 805.13  ; #2扫码位有料感应标志[0005.13]
ANDNOT H11.00  ; #1隔离气缸放料中记忆
ANDNOT H13.00  ; #2隔离气缸放料中记忆
AND 10.03  ; #1隔离气缸伸出
AND 10.07  ; #2隔离气缸伸出
ORLD
LD D1006.04  ; 进料拉带机构扫码触发（步）
LD W65.02  ; 进料#1扫码失败
LD W75.02  ; 进料#2扫码失败
OR W75.03  ; 进料#2扫码成功
ANDLD
LD W65.03  ; 进料#1扫码成功
AND W75.02  ; 进料#2扫码失败
ORLD
LD H10.06  ; #1扫码阻挡扫码完成记忆
AND H12.06  ; #2扫码阻挡扫码完成记忆
ORLD
ANDLD
ORLD
LD D1006.05  ; 进料拉带机构扫码结果（步）
AND H10.06  ; #1扫码阻挡扫码完成记忆
AND H12.06  ; #2扫码阻挡扫码完成记忆
ORLD
LD D1006.06  ; 进料拉带机构扫码MES入站校验结果（步）
LD H10.09  ; #1扫码阻挡MES校验完成记忆
OR H10.08  ; #1扫码阻挡扫码NG料记忆
ANDLD
LD H12.09  ; #2扫码阻挡MES校验完成记忆
OR H12.08  ; #2扫码阻挡扫码NG料记忆
ANDLD
AND H10.06  ; #1扫码阻挡扫码完成记忆
AND H12.06  ; #2扫码阻挡扫码完成记忆
AND H10.00  ; #1扫码阻挡有料记忆
AND H12.00  ; #2扫码阻挡有料记忆
AND D1001.02  ; 进料拉带扫码阻挡气缸允许放料条件
ORLD
OR D1006.07  ; 预留
LD D1006.08  ; 进料拉带机构扫码阻挡气缸缩回&进料拉带电机启动（步）
AND 800.00  ; #1扫码阻挡气缸缩回位标志[0000.00]
AND 800.04  ; #2扫码阻挡气缸缩回位标志[0000.04]
LD 15.00  ; 进料拉带电机启动
OR P_On
ANDLD
ANDNOT H10.00  ; #1扫码阻挡有料记忆
ANDNOT 805.12  ; #1扫码位有料感应标志[0005.12]
ANDNOT H12.00  ; #2扫码阻挡有料记忆
ANDNOT 805.13  ; #2扫码位有料感应标志[0005.13]
LD H10.01  ; #1进料位有料记忆
AND H12.01  ; #2进料位有料记忆
AND 805.15  ; #1-2进料位有料感应标志[0005.15]
AND 806.01  ; #2-2进料位有料感应标志[0006.01]
ORNOT P_On
ANDLD
ANDNOT H11.01  ; #1扫码阻挡气缸放料中记忆
ANDNOT H13.01  ; #2扫码阻挡气缸放料中记忆
ORLD
LD D1006.09  ; 进料拉带机构扫码阻挡气缸伸出（步）
AND 800.01  ; #1扫码阻挡气缸伸出位标志[0000.01]
AND 800.05  ; #2扫码阻挡气缸伸出位标志[0000.05]
ORLD
OR D1006.10  ; 预留
LD D1004.01  ; 进料拉带机构单步/自动循环运行中
AND W1.01  ; 自动模式
@LD D1003.15  ; 进料拉带机构单步（SW）
AND D1004.10  ; 进料拉带机构单步运行条件
ORLD
ANDLD
OUT D1005.01  ; 进料拉带机构步进条件

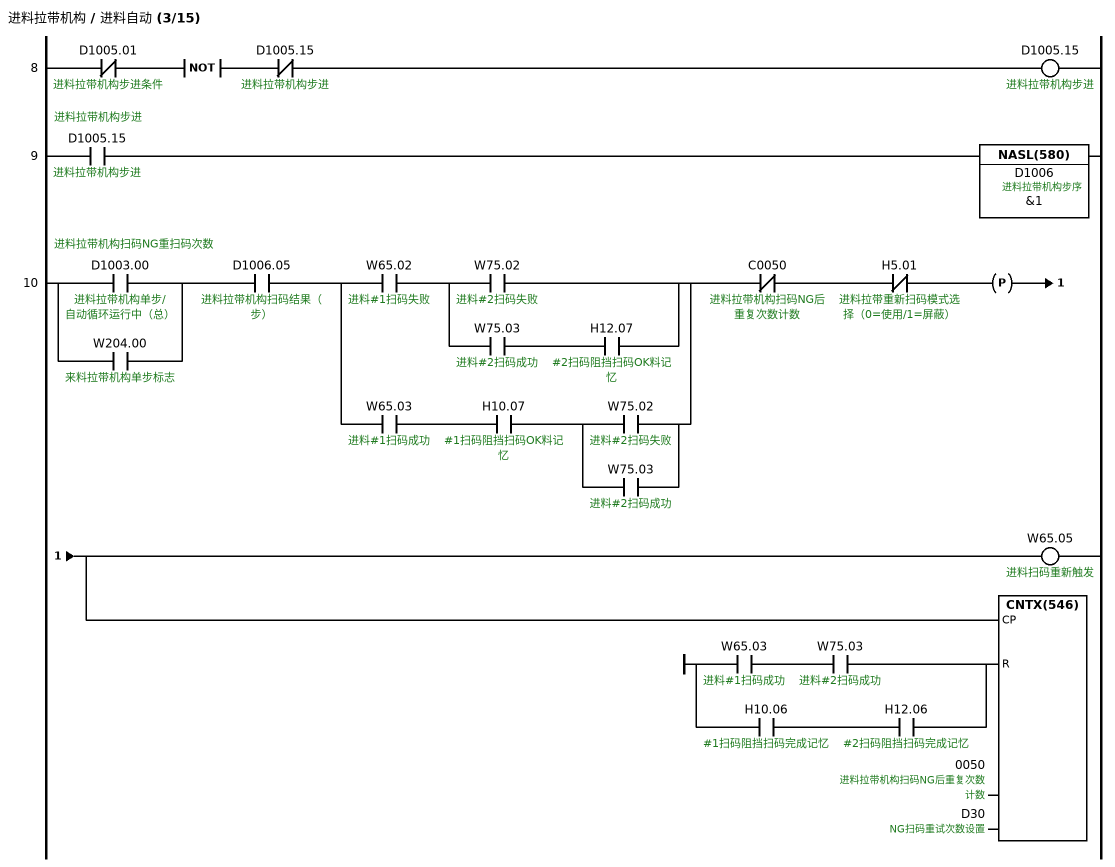
; rung 8
LDNOT D1005.01  ; 进料拉带机构步进条件
NOT(520)
ANDNOT D1005.15  ; 进料拉带机构步进
OUT D1005.15  ; 进料拉带机构步进
; rung 9: 进料拉带机构步进
LD D1005.15  ; 进料拉带机构步进
NASL(580) D1006 &1  ; 进料拉带机构步序
; rung 10: 进料拉带机构扫码NG重扫码次数
LD D1003.00  ; 进料拉带机构单步/自动循环运行中（总）
OR W204.00  ; 来料拉带机构单步标志
AND D1006.05  ; 进料拉带机构扫码结果（步）
LD W65.02  ; 进料#1扫码失败
LD W75.02  ; 进料#2扫码失败
LD W75.03  ; 进料#2扫码成功
AND H12.07  ; #2扫码阻挡扫码OK料记忆
ORLD
ANDLD
LD W65.03  ; 进料#1扫码成功
AND H10.07  ; #1扫码阻挡扫码OK料记忆
LD W75.02  ; 进料#2扫码失败
OR W75.03  ; 进料#2扫码成功
ANDLD
ORLD
ANDLD
ANDNOT C0050  ; 进料拉带机构扫码NG后重复次数计数
ANDNOT H5.01  ; 进料拉带重新扫码模式选择（0=使用/1=屏蔽）
UP(521)
OUT W65.05  ; 进料扫码重新触发
LD W65.03  ; 进料#1扫码成功
AND W75.03  ; 进料#2扫码成功
LD H10.06  ; #1扫码阻挡扫码完成记忆
AND H12.06  ; #2扫码阻挡扫码完成记忆
ORLD
CNTX(546) 0050 D30  ; NG扫码重试次数设置, 进料拉带机构扫码NG后重复次数计数

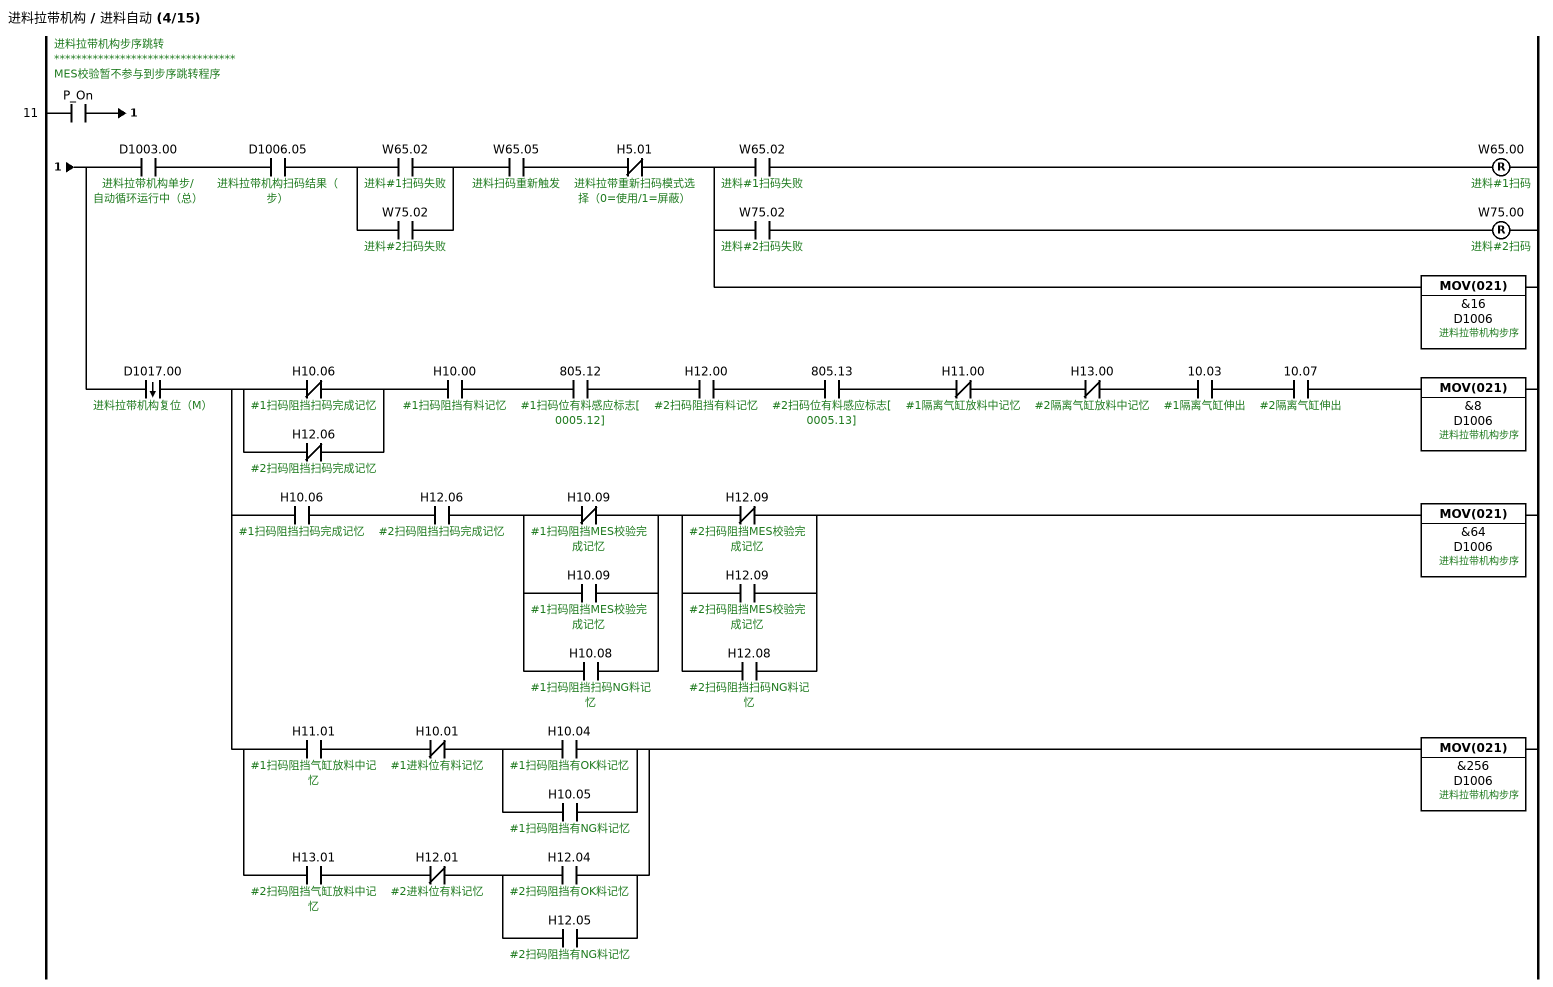
; rung 11: 进料拉带机构步序跳转 / ********************************* / MES校验暂不参与到步序跳转程序
LD P_On
OUT TR0
AND D1003.00  ; 进料拉带机构单步/自动循环运行中（总）
AND D1006.05  ; 进料拉带机构扫码结果（步）
LD W65.02  ; 进料#1扫码失败
OR W75.02  ; 进料#2扫码失败
ANDLD
AND W65.05  ; 进料扫码重新触发
ANDNOT H5.01  ; 进料拉带重新扫码模式选择（0=使用/1=屏蔽）
OUT TR1
AND W65.02  ; 进料#1扫码失败
RSET W65.00  ; 进料#1扫码
LD TR1
AND W75.02  ; 进料#2扫码失败
RSET W75.00  ; 进料#2扫码
LD TR1
MOV(021) &16 D1006  ; 进料拉带机构步序  // 进料拉带机构扫码触发步（D1006.04）
LD TR0
%AND D1017.00  ; 进料拉带机构复位（M）
OUT TR0
LDNOT H10.06  ; #1扫码阻挡扫码完成记忆
ORNOT H12.06  ; #2扫码阻挡扫码完成记忆
ANDLD
AND H10.00  ; #1扫码阻挡有料记忆
AND 805.12  ; #1扫码位有料感应标志[0005.12]
AND H12.00  ; #2扫码阻挡有料记忆
AND 805.13  ; #2扫码位有料感应标志[0005.13]
ANDNOT H11.00  ; #1隔离气缸放料中记忆
ANDNOT H13.00  ; #2隔离气缸放料中记忆
AND 10.03  ; #1隔离气缸伸出
AND 10.07  ; #2隔离气缸伸出
MOV(021) &8 D1006  ; 进料拉带机构步序  // 进料拉带机构扫码触发前延时步（D1006.03）
LD TR0
AND H10.06  ; #1扫码阻挡扫码完成记忆
AND H12.06  ; #2扫码阻挡扫码完成记忆
LDNOT H10.09  ; #1扫码阻挡MES校验完成记忆
OR H10.09  ; #1扫码阻挡MES校验完成记忆
OR H10.08  ; #1扫码阻挡扫码NG料记忆
ANDLD
LDNOT H12.09  ; #2扫码阻挡MES校验完成记忆
OR H12.09  ; #2扫码阻挡MES校验完成记忆
OR H12.08  ; #2扫码阻挡扫码NG料记忆
ANDLD
MOV(021) &64 D1006  ; 进料拉带机构步序  // 进料拉带机构扫码MES入站校验结果步（D1006.06）
LD TR0
LD H11.01  ; #1扫码阻挡气缸放料中记忆
ANDNOT H10.01  ; #1进料位有料记忆
LD H10.04  ; #1扫码阻挡有OK料记忆
OR H10.05  ; #1扫码阻挡有NG料记忆
ANDLD
LD H13.01  ; #2扫码阻挡气缸放料中记忆
ANDNOT H12.01  ; #2进料位有料记忆
LD H12.04  ; #2扫码阻挡有OK料记忆
OR H12.05  ; #2扫码阻挡有NG料记忆
ANDLD
ORLD
ANDLD
MOV(021) &256 D1006  ; 进料拉带机构步序  // 进料拉带机构扫码阻挡气缸缩回&进料拉带电机启动步（D1006.08）

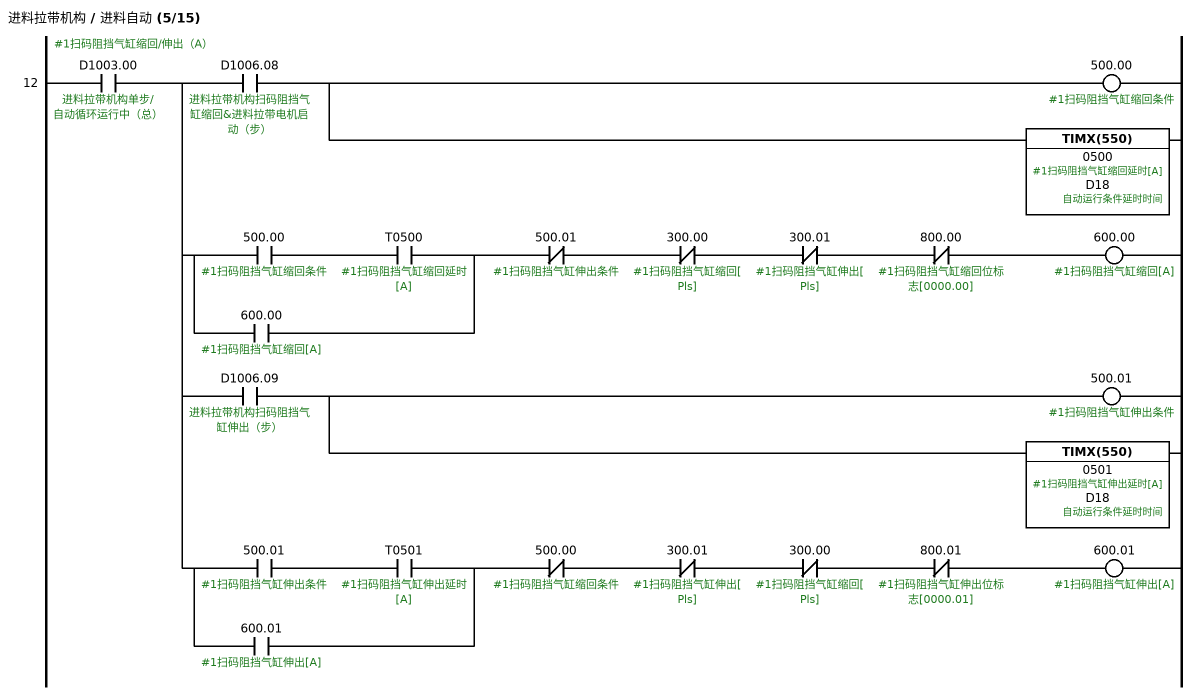
; rung 12: #1扫码阻挡气缸缩回/伸出（A）
LD D1003.00  ; 进料拉带机构单步/自动循环运行中（总）
OUT TR0
AND D1006.08  ; 进料拉带机构扫码阻挡气缸缩回&进料拉带电机启动（步）
OUT 500.00  ; #1扫码阻挡气缸缩回条件
TIMX(550) 0500 D18  ; 自动运行条件延时时间, #1扫码阻挡气缸缩回延时[A]
LD TR0
LD 500.00  ; #1扫码阻挡气缸缩回条件
AND T0500  ; #1扫码阻挡气缸缩回延时[A]
OR 600.00  ; #1扫码阻挡气缸缩回[A]
ANDLD
ANDNOT 500.01  ; #1扫码阻挡气缸伸出条件
ANDNOT 300.00  ; #1扫码阻挡气缸缩回[Pls]
ANDNOT 300.01  ; #1扫码阻挡气缸伸出[Pls]
ANDNOT 800.00  ; #1扫码阻挡气缸缩回位标志[0000.00]
OUT 600.00  ; #1扫码阻挡气缸缩回[A]
LD TR0
AND D1006.09  ; 进料拉带机构扫码阻挡气缸伸出（步）
OUT 500.01  ; #1扫码阻挡气缸伸出条件
TIMX(550) 0501 D18  ; 自动运行条件延时时间, #1扫码阻挡气缸伸出延时[A]
LD TR0
LD 500.01  ; #1扫码阻挡气缸伸出条件
AND T0501  ; #1扫码阻挡气缸伸出延时[A]
OR 600.01  ; #1扫码阻挡气缸伸出[A]
ANDLD
ANDNOT 500.00  ; #1扫码阻挡气缸缩回条件
ANDNOT 300.01  ; #1扫码阻挡气缸伸出[Pls]
ANDNOT 300.00  ; #1扫码阻挡气缸缩回[Pls]
ANDNOT 800.01  ; #1扫码阻挡气缸伸出位标志[0000.01]
OUT 600.01  ; #1扫码阻挡气缸伸出[A]

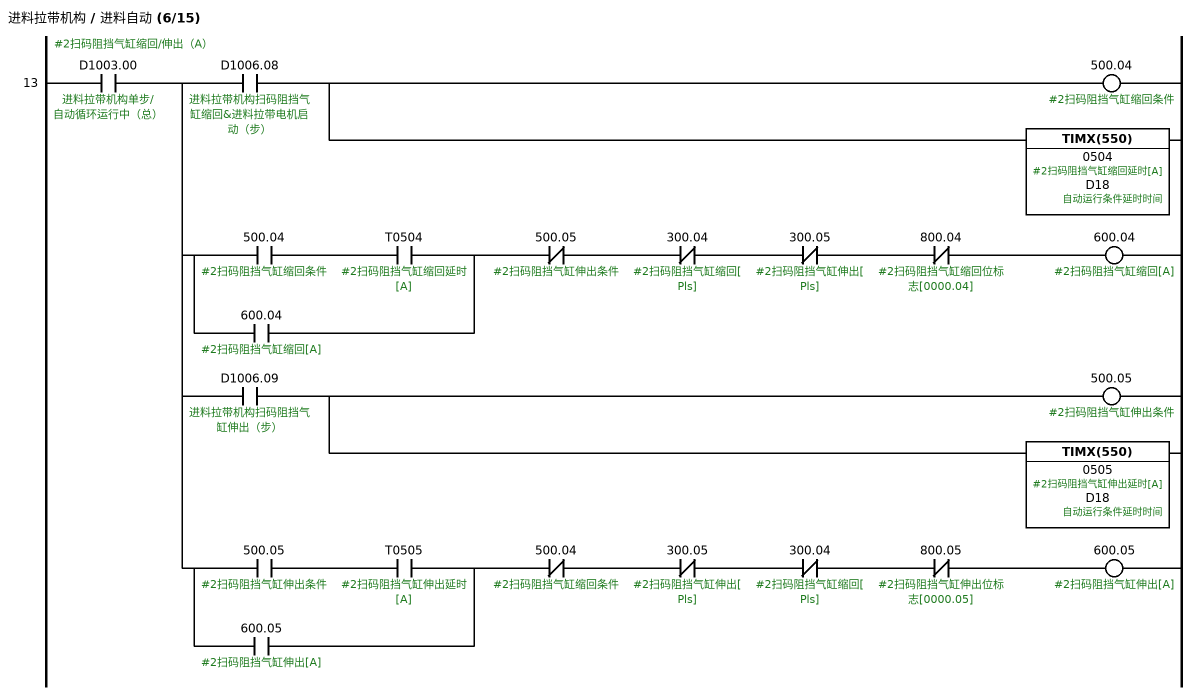
; rung 13: #2扫码阻挡气缸缩回/伸出（A）
LD D1003.00  ; 进料拉带机构单步/自动循环运行中（总）
OUT TR0
AND D1006.08  ; 进料拉带机构扫码阻挡气缸缩回&进料拉带电机启动（步）
OUT 500.04  ; #2扫码阻挡气缸缩回条件
TIMX(550) 0504 D18  ; 自动运行条件延时时间, #2扫码阻挡气缸缩回延时[A]
LD TR0
LD 500.04  ; #2扫码阻挡气缸缩回条件
AND T0504  ; #2扫码阻挡气缸缩回延时[A]
OR 600.04  ; #2扫码阻挡气缸缩回[A]
ANDLD
ANDNOT 500.05  ; #2扫码阻挡气缸伸出条件
ANDNOT 300.04  ; #2扫码阻挡气缸缩回[Pls]
ANDNOT 300.05  ; #2扫码阻挡气缸伸出[Pls]
ANDNOT 800.04  ; #2扫码阻挡气缸缩回位标志[0000.04]
OUT 600.04  ; #2扫码阻挡气缸缩回[A]
LD TR0
AND D1006.09  ; 进料拉带机构扫码阻挡气缸伸出（步）
OUT 500.05  ; #2扫码阻挡气缸伸出条件
TIMX(550) 0505 D18  ; 自动运行条件延时时间, #2扫码阻挡气缸伸出延时[A]
LD TR0
LD 500.05  ; #2扫码阻挡气缸伸出条件
AND T0505  ; #2扫码阻挡气缸伸出延时[A]
OR 600.05  ; #2扫码阻挡气缸伸出[A]
ANDLD
ANDNOT 500.04  ; #2扫码阻挡气缸缩回条件
ANDNOT 300.05  ; #2扫码阻挡气缸伸出[Pls]
ANDNOT 300.04  ; #2扫码阻挡气缸缩回[Pls]
ANDNOT 800.05  ; #2扫码阻挡气缸伸出位标志[0000.05]
OUT 600.05  ; #2扫码阻挡气缸伸出[A]

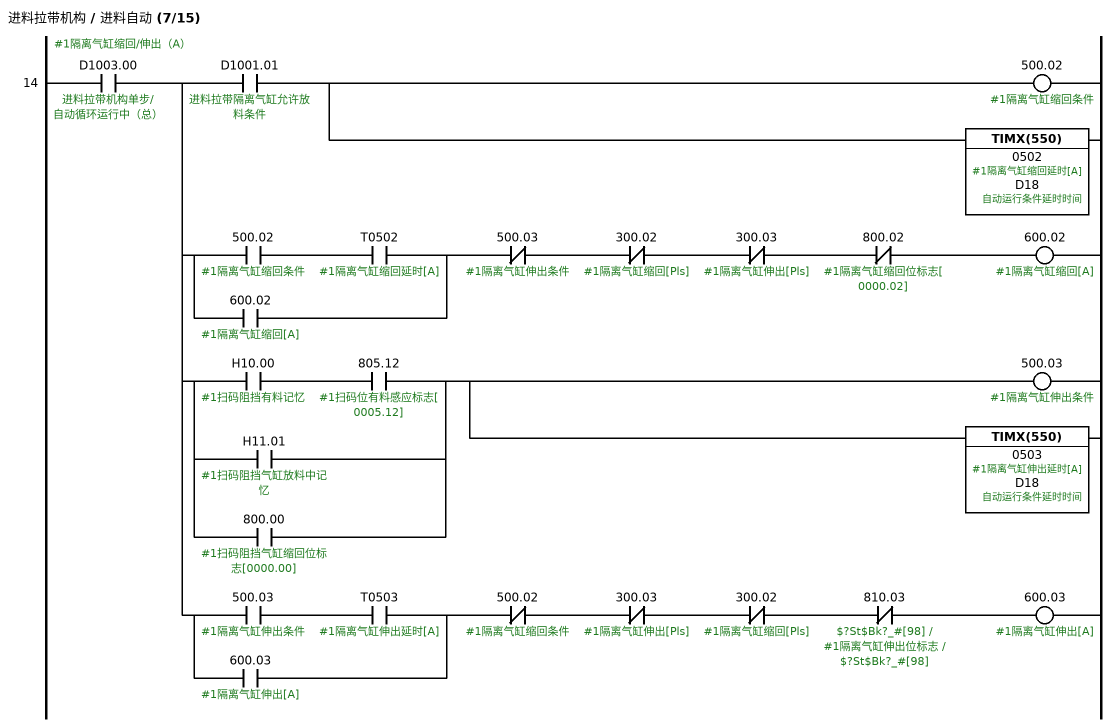
; rung 14: #1隔离气缸缩回/伸出（A）
LD D1003.00  ; 进料拉带机构单步/自动循环运行中（总）
OUT TR0
AND D1001.01  ; 进料拉带隔离气缸允许放料条件
OUT 500.02  ; #1隔离气缸缩回条件
TIMX(550) 0502 D18  ; 自动运行条件延时时间, #1隔离气缸缩回延时[A]
LD TR0
LD 500.02  ; #1隔离气缸缩回条件
AND T0502  ; #1隔离气缸缩回延时[A]
OR 600.02  ; #1隔离气缸缩回[A]
ANDLD
ANDNOT 500.03  ; #1隔离气缸伸出条件
ANDNOT 300.02  ; #1隔离气缸缩回[Pls]
ANDNOT 300.03  ; #1隔离气缸伸出[Pls]
ANDNOT 800.02  ; #1隔离气缸缩回位标志[0000.02]
OUT 600.02  ; #1隔离气缸缩回[A]
LD TR0
LD H10.00  ; #1扫码阻挡有料记忆
AND 805.12  ; #1扫码位有料感应标志[0005.12]
OR H11.01  ; #1扫码阻挡气缸放料中记忆
OR 800.00  ; #1扫码阻挡气缸缩回位标志[0000.00]
ANDLD
OUT 500.03  ; #1隔离气缸伸出条件
TIMX(550) 0503 D18  ; 自动运行条件延时时间, #1隔离气缸伸出延时[A]
LD TR0
LD 500.03  ; #1隔离气缸伸出条件
AND T0503  ; #1隔离气缸伸出延时[A]
OR 600.03  ; #1隔离气缸伸出[A]
ANDLD
ANDNOT 500.02  ; #1隔离气缸缩回条件
ANDNOT 300.03  ; #1隔离气缸伸出[Pls]
ANDNOT 300.02  ; #1隔离气缸缩回[Pls]
ANDNOT 810.03  ; $?St$Bk?_#[98] / #1隔离气缸伸出位标志 / $?St$Bk?_#[98]
OUT 600.03  ; #1隔离气缸伸出[A]

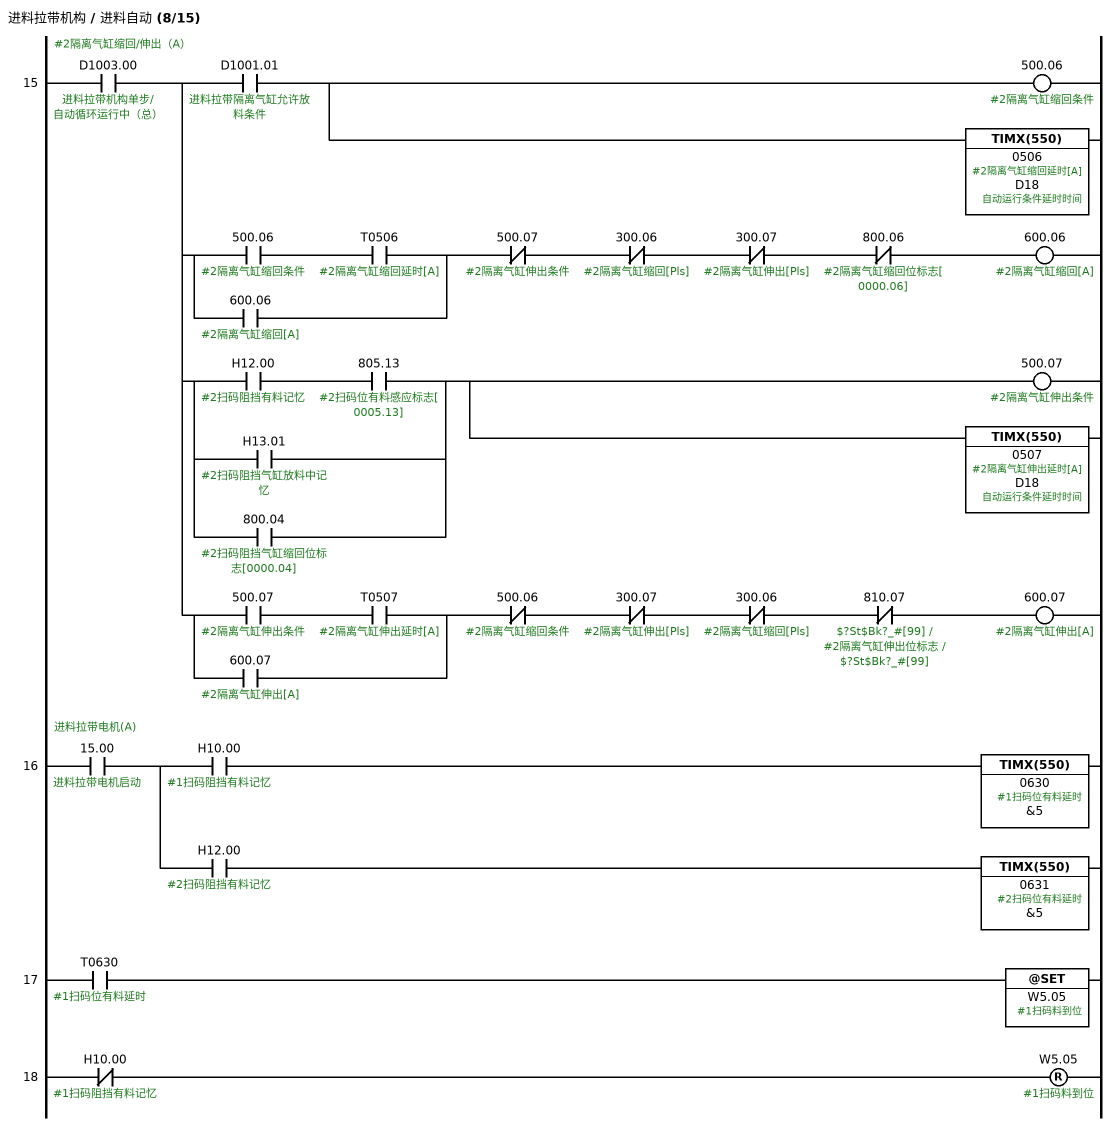
; rung 15: #2隔离气缸缩回/伸出（A）
LD D1003.00  ; 进料拉带机构单步/自动循环运行中（总）
OUT TR0
AND D1001.01  ; 进料拉带隔离气缸允许放料条件
OUT 500.06  ; #2隔离气缸缩回条件
TIMX(550) 0506 D18  ; 自动运行条件延时时间, #2隔离气缸缩回延时[A]
LD TR0
LD 500.06  ; #2隔离气缸缩回条件
AND T0506  ; #2隔离气缸缩回延时[A]
OR 600.06  ; #2隔离气缸缩回[A]
ANDLD
ANDNOT 500.07  ; #2隔离气缸伸出条件
ANDNOT 300.06  ; #2隔离气缸缩回[Pls]
ANDNOT 300.07  ; #2隔离气缸伸出[Pls]
ANDNOT 800.06  ; #2隔离气缸缩回位标志[0000.06]
OUT 600.06  ; #2隔离气缸缩回[A]
LD TR0
LD H12.00  ; #2扫码阻挡有料记忆
AND 805.13  ; #2扫码位有料感应标志[0005.13]
OR H13.01  ; #2扫码阻挡气缸放料中记忆
OR 800.04  ; #2扫码阻挡气缸缩回位标志[0000.04]
ANDLD
OUT 500.07  ; #2隔离气缸伸出条件
TIMX(550) 0507 D18  ; 自动运行条件延时时间, #2隔离气缸伸出延时[A]
LD TR0
LD 500.07  ; #2隔离气缸伸出条件
AND T0507  ; #2隔离气缸伸出延时[A]
OR 600.07  ; #2隔离气缸伸出[A]
ANDLD
ANDNOT 500.06  ; #2隔离气缸缩回条件
ANDNOT 300.07  ; #2隔离气缸伸出[Pls]
ANDNOT 300.06  ; #2隔离气缸缩回[Pls]
ANDNOT 810.07  ; $?St$Bk?_#[99] / #2隔离气缸伸出位标志 / $?St$Bk?_#[99]
OUT 600.07  ; #2隔离气缸伸出[A]
; rung 16: 进料拉带电机(A)
LD 15.00  ; 进料拉带电机启动
OUT TR0
AND H10.00  ; #1扫码阻挡有料记忆
TIMX(550) 0630 &5  ; #1扫码位有料延时
LD TR0
AND H12.00  ; #2扫码阻挡有料记忆
TIMX(550) 0631 &5  ; #2扫码位有料延时
; rung 17
LD T0630  ; #1扫码位有料延时
@SET W5.05  ; #1扫码料到位
; rung 18
LDNOT H10.00  ; #1扫码阻挡有料记忆
RSET W5.05  ; #1扫码料到位

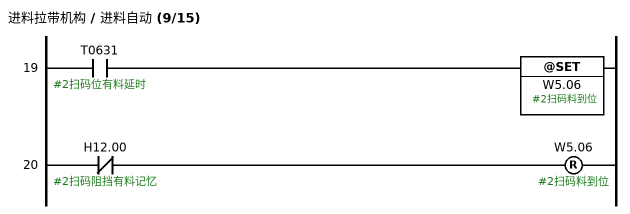
; rung 19
LD T0631  ; #2扫码位有料延时
@SET W5.06  ; #2扫码料到位
; rung 20
LDNOT H12.00  ; #2扫码阻挡有料记忆
RSET W5.06  ; #2扫码料到位

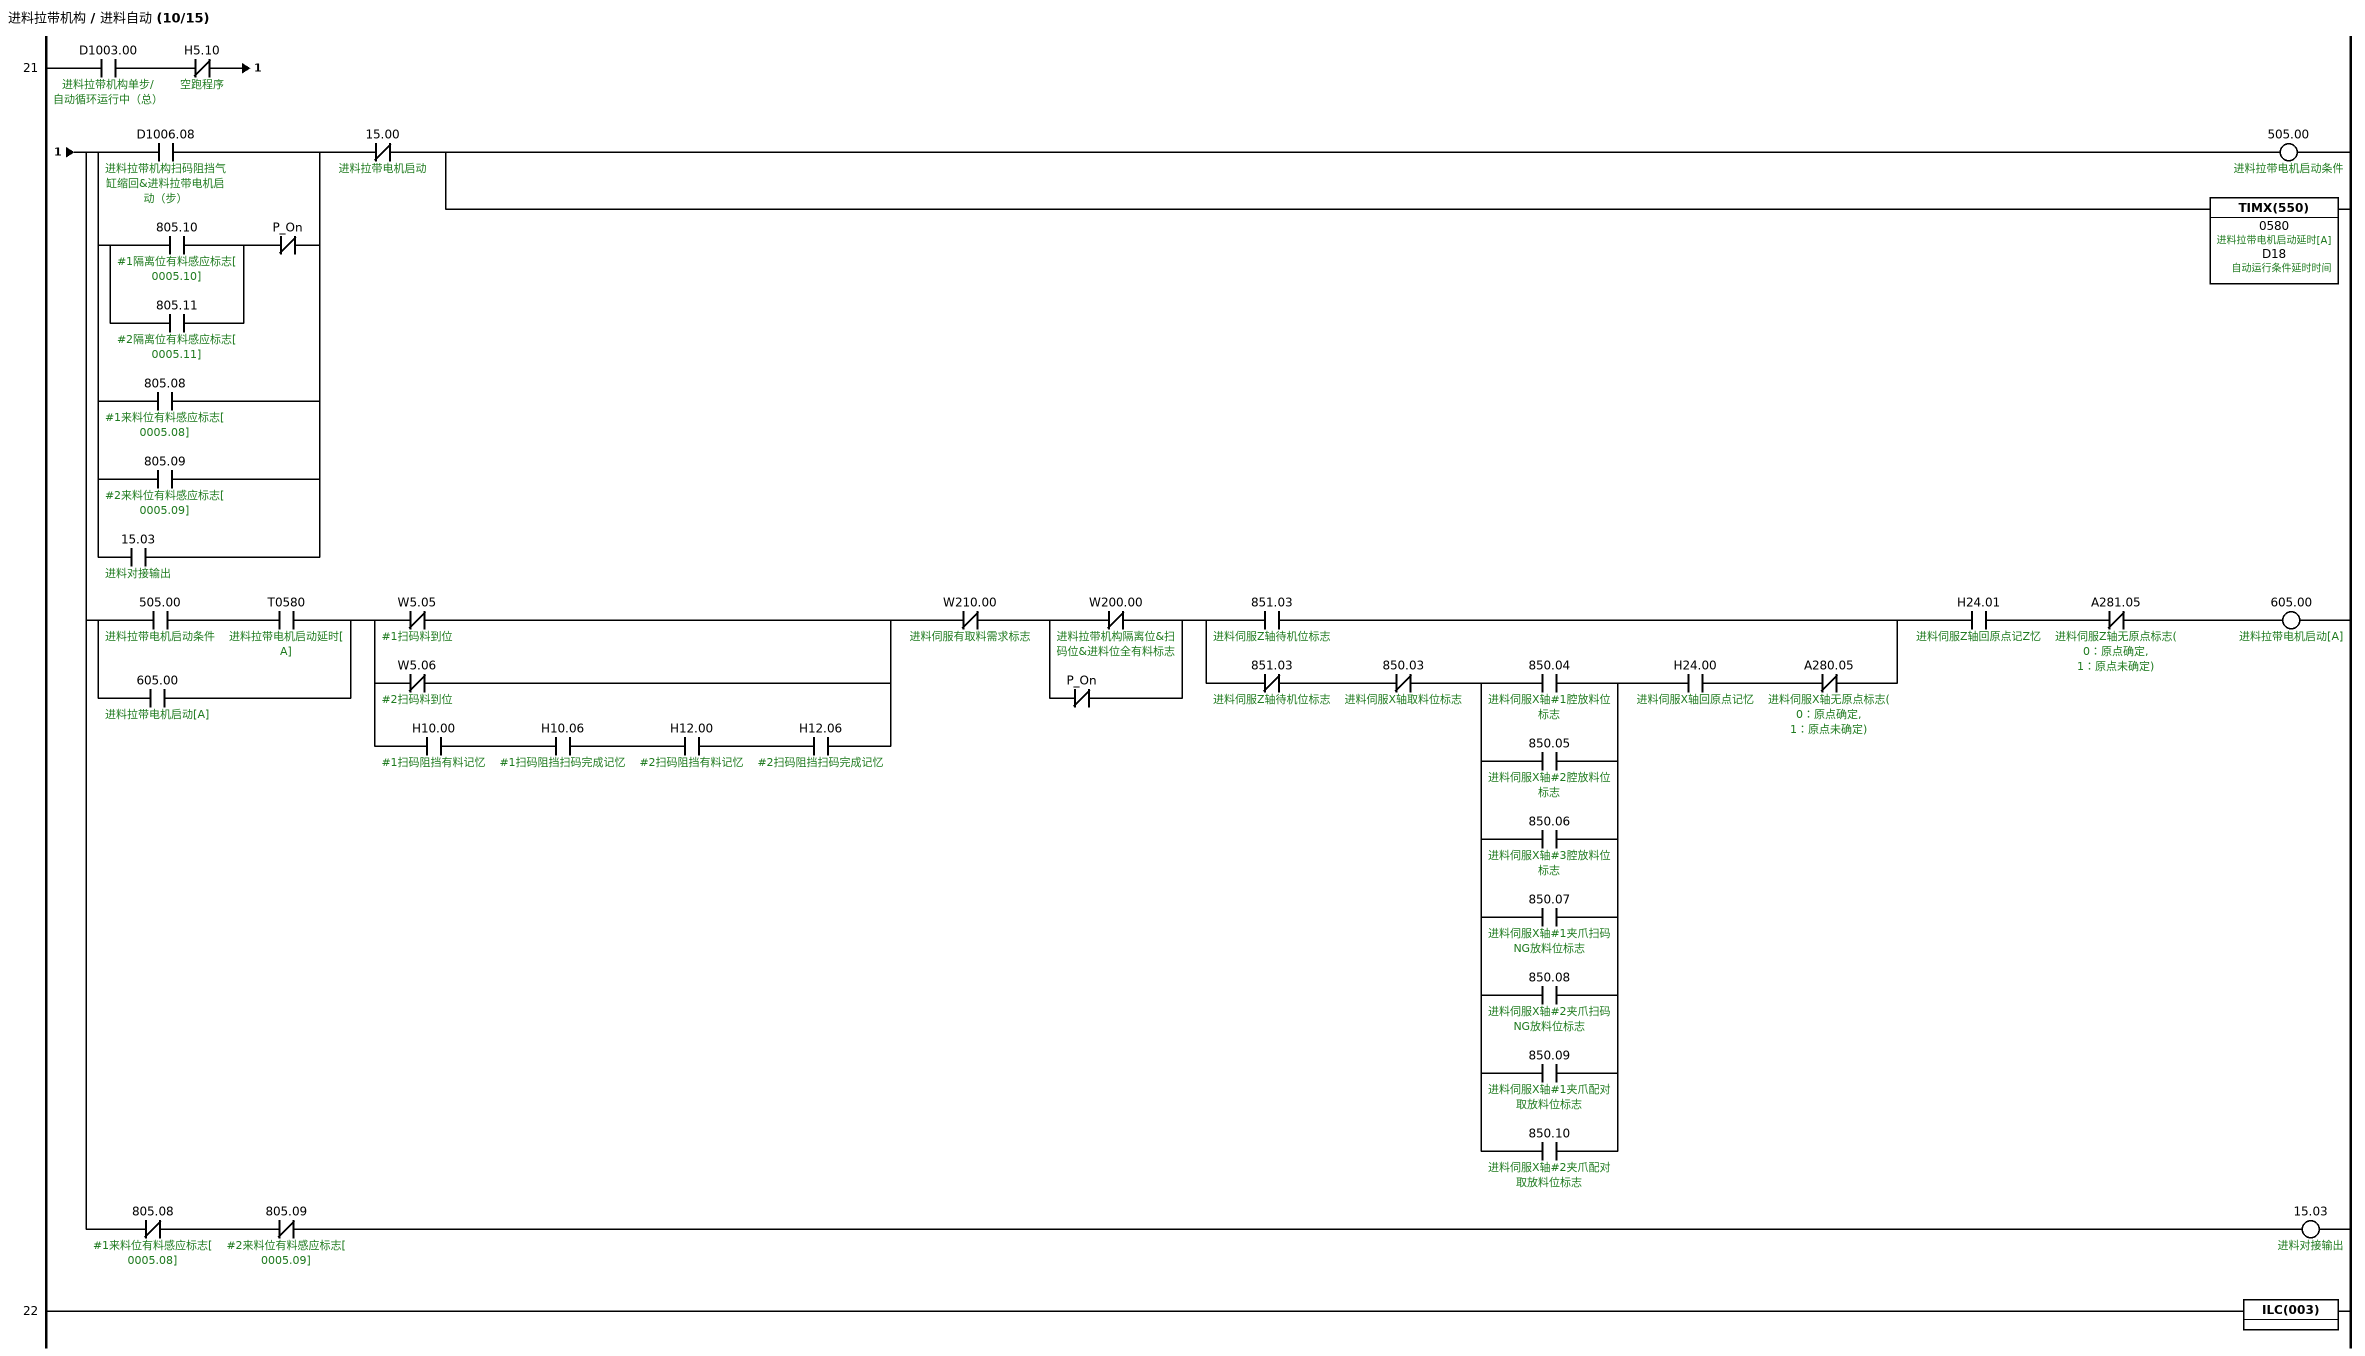
; rung 21
LD D1003.00  ; 进料拉带机构单步/自动循环运行中（总）
ANDNOT H5.10  ; 空跑程序
OUT TR0
LD D1006.08  ; 进料拉带机构扫码阻挡气缸缩回&进料拉带电机启动（步）
LD 805.10  ; #1隔离位有料感应标志[0005.10]
OR 805.11  ; #2隔离位有料感应标志[0005.11]
ANDNOT P_On
ORLD
OR 805.08  ; #1来料位有料感应标志[0005.08]
OR 805.09  ; #2来料位有料感应标志[0005.09]
OR 15.03  ; 进料对接输出  // 允许上工位放料
ANDLD
ANDNOT 15.00  ; 进料拉带电机启动
OUT 505.00  ; 进料拉带电机启动条件
TIMX(550) 0580 D18  ; 自动运行条件延时时间, 进料拉带电机启动延时[A]
LD TR0
LD 505.00  ; 进料拉带电机启动条件
AND T0580  ; 进料拉带电机启动延时[A]
OR 605.00  ; 进料拉带电机启动[A]
ANDLD
LDNOT W5.05  ; #1扫码料到位
ORNOT W5.06  ; #2扫码料到位
LD H10.00  ; #1扫码阻挡有料记忆
AND H10.06  ; #1扫码阻挡扫码完成记忆  // 省略#1扫码MES校验完成记忆
AND H12.00  ; #2扫码阻挡有料记忆
AND H12.06  ; #2扫码阻挡扫码完成记忆  // 省略#2扫码MES校验完成记忆
ORLD
ANDLD
ANDNOT W210.00  ; 进料伺服有取料需求标志
LDNOT W200.00  ; 进料拉带机构隔离位&扫码位&进料位全有料标志
ORNOT P_On
ANDLD
LD 851.03  ; 进料伺服Z轴待机位标志
LDNOT 851.03  ; 进料伺服Z轴待机位标志
ANDNOT 850.03  ; 进料伺服X轴取料位标志
LD 850.04  ; 进料伺服X轴#1腔放料位标志
OR 850.05  ; 进料伺服X轴#2腔放料位标志
OR 850.06  ; 进料伺服X轴#3腔放料位标志
OR 850.07  ; 进料伺服X轴#1夹爪扫码NG放料位标志
OR 850.08  ; 进料伺服X轴#2夹爪扫码NG放料位标志
OR 850.09  ; 进料伺服X轴#1夹爪配对取放料位标志
OR 850.10  ; 进料伺服X轴#2夹爪配对取放料位标志
ANDLD
AND H24.00  ; 进料伺服X轴回原点记忆
ANDNOT A280.05  ; 进料伺服X轴无原点标志(0：原点确定,1：原点未确定)
ORLD
ANDLD
AND H24.01  ; 进料伺服Z轴回原点记Z忆
ANDNOT A281.05  ; 进料伺服Z轴无原点标志(0：原点确定,1：原点未确定)
OUT 605.00  ; 进料拉带电机启动[A]
LD TR0
ANDNOT 805.08  ; #1来料位有料感应标志[0005.08]
ANDNOT 805.09  ; #2来料位有料感应标志[0005.09]
OUT 15.03  ; 进料对接输出
; rung 22
ILC(003)

